(* Logix 5000 project; controller cal1615 1756-L62 rev 20.19; software revision 20.05; part 6 of 81 *)

        [13]   // Advanced Cooling Real to HMI Analog Input Recirc Fan Amps
        [14]   // Advanced Cooling Real to HMI Analog Analog Input Recirc Fan RPM
        [15]   // Advanced Cooling Real to HMI Analog Analog Input Recirc Fan Pct
        [16]   // Advanced Cooling Real to HMI Analog Input Spare
        [17]   // Advanced Cooling Real to HMI Analog Input Spare
        [24]   // Advanced Cooling Real to HMI Analog Output Hot Air Damper
        [28]   // Advanced Cooling Real to HMI Analog Output Exhaust Fan VFD Selected Speed
        [30]   // Advanced Cooling Real to HMI Analog Output Supply Fan VFD Selected Speed
        [40]   // Advanced Cooling Real to HMI Parameter TC01 Temperature Zero Offset
        [41]   // Advanced Cooling Real to HMI Parameter TC02 Temperature Zero Offset
        [42]   // Advanced Cooling Real to HMI Parameter
        [43]   // Advanced Cooling Real to HMI Parameter
        [44]   // Advanced Cooling Real to HMI Parameter PID1 NKp
        [45]   // Advanced Cooling Real to HMI Parameter PID1 Ki
        [46]   // Advanced Cooling Real to HMI Parameter PID1 Kd
        [47]   // Advanced Cooling Real to HMI Parameter PID1 Bias
        [48]   // Advanced Cooling Real to HMI Parameter PID2 Kp
        [49]   // Advanced Cooling Real to HMI Parameter PID2 Ki
        [50]   // Advanced Cooling Real to HMI Parameter PID2 Kd
        [51]   // Advanced Cooling Real to HMI Parameter PID2 Bias
        [52]   // Advanced Cooling Real to HMI Parameter Process Control High Limit
        [53]   // Advanced Cooling Real to HMI Parameter Spare
        [54]   // Advanced Cooling Real to HMI parameter Process Control Deviation
        [55]   // Advanced Cooling Real to HMI Parameter LFL Warning Level
        [56]   // Advanced Cooling Real to HMI Parameter LFL Alarm Level
        [57]   // Advanced Cooling Real to HMI Parameter Zone Shutdown Temperature
        [58]   // Advanced Cooling Real to HMI Parameter High Pressure LImit
        [59]   // Advanced Cooling Real to HMI Temperature Control Fast to Soak Control Deviation
        [60]   // Advanced Cooling Real to HMI Temperature Control Soak to Fast Control Deviation
        [61]   // Advanced Cooling Real to HMI Parameter
        [62]   // Advanced Cooling Real to HMI Parameter
        [63]   // Advanced Cooling Real to HMI Parameter
        [64]   // Advanced Cooling Real to HMI Exhaust VFD RPM Setpoint
        [65]   // Advanced Cooling Real to HMI Recirc VFD RPM Setpoint
        [67]   // Advanced Cooling Real to HMI Temperature Control Setpoint
        [68]   // Advanced Cooling Real to HMI Temperature Control manual Control Valve Setpoint
        [69]   // Advanced Cooling Real to HMI
        [70]   // Advanced Cooling Real to HMI
        [71]   // Advanced Cooling Real to HMI
        [72]   // Advanced Cooling Real to HMI Process Control Temperature
        [73]   // Advanced Cooling Real to HMI
        [74]   // Advanced Cooling Real to HMI
        [75]   // Advanced Cooling Real to HMI
        [76]   // Advanced Cooling Real to HMI
        [77]   // Advanced Cooling Real to HMI
        [78]   // Advanced Cooling Real to HMI
        [79]   // Advanced Cooling Real to HMI
   p19r01 : routine := (comment := 7);   // Advanced Cooling Main
   p19r02 : routine := (comment := -1073741761);   // Advanced Cooling Misc Control
        .WARNING.0   // Advanced Cooling Misc Control Warning 0
   p19r02_fault_exists : BOOL;
   p19r02_timer_fault : TIMER[4];   // Advanced Cooling Misc Control Fault Delay
   p19r02_timer_warning : TIMER[4] := ([0].PRE := 1500);   // Advanced Cooling Warning Delay
   p19r02_unack_fault : BOOL;   // Advanced Cooling Misc Control Unacknowledged Fault
   p19r02_unack_warning : BOOL;   // Advanced Cooling Misc Control Unacknowledged Warning
   p19r02_warning_exists : BOOL;
   p19r03 : routine := (comment := -1073741761);   // Advanced Cooling Input
   p19r03_flow_scp : SYS_SCP := (Input_Max := 100.0, Output_Max := 30840.0);   // Advanced Cooling Output Roll Cooling Flow Control
   p19r03_prs_input_max : REAL := 30840.0;
   p19r03_prs_input_min : REAL;
   p19r03_prs_output_max : REAL := 50.0;
   p19r03_prs_output_min : REAL;
   p19r03_prs_scp : SYS_SCP := (Input := 60.0, Input_Max := 100.0, Output_Max := 30840.0, Output := 18504.0);   // Advanced Cooling Output Cooling Pressure Control Valve Output
   p19r03_timer_fault : TIMER[4];   // Advanced Cooling Input
   p19r03_timer_warning : TIMER[4];   // Advanced Cooling Input
   p19r04 : routine := (comment := -1073741761);   // Advanced Cooling Output
   p19r04_timer_fault : TIMER[4];   // Advanced Cooling Output Fault Delay
   p19r04_timer_warning : TIMER[4];   // Advanced Cooling Output Warning Delay
   p19r05 : routine := (comment := -1073741761);   // Advanced Cooling Dint to HMI
   p19r05_timer_fault : TIMER[4];   // Advanced Cooing Dint to HMI
   p19r05_timer_warning : TIMER[4];   // Advanced Cooling Dint to HMI Warning Delay
   p19r06 : routine := (comment := -1073741572);   // Advanced Cooling Real to HMI
   p19r06_timer_fault : TIMER[4];   // Advanced Cooling Real to HMI Fault Delay
   p19r06_timer_warning : TIMER[4];   // Advanced Cooling Real to HMI Warning Delay
   p19r07 : routine := (comment := -1073741761);   // Advanced Cooling Alarms
   p19r07_timer_fault : TIMER[4];   // Advanced Cooling Alarms Fault Delay
   p19r07_timer_warning : TIMER[4];   // Advanced Cooling Alarms Warning Delay
   p19r08 : routine := (comment := -1073741761);   // Advanced Cooling Warnings
   p19r08_timer_fault : TIMER[4];   // Advanced Cooling Warnings Fault Delay
   p19r08_timer_warning : TIMER[4];   // Advanced Cooling Warnings Warning Delay
   p19r09 : routine := (comment := -1073741761);   // Advanced Cooling Modes
   p19r09_timer_fault : TIMER[4];   // Advanced Cooling Modes Fault Delay
   p19r09_timer_warning : TIMER[4];   // Advanced Cooling Modes Warning Delay
   p19r10 : routine := (comment := -1073741761);   // Advanced Cooling Parameters
   p19r10_timer_fault : TIMER[4];   // Advanced Cooling Parameters Fault Delay
   p19r10_timer_warning : TIMER[4];   // Advanced Cooling Parameters Warning Delay
   p19r16_pid_temp_cv : DINT;   // Advanced Cooling Temperature Control PID Control Valve
   p19r30 : routine := (comment := -1073741697);   // Advanced Cooling Temperature Control
        .FAULT.2   // Advanced Cooling Temperature Control Thermocouple Failure
        .WARNING.0   // Advanced Cooling Temperature Control Temperature Deviation Warning
        .WARNING.1   // Advanced Cooling Temperature Control Control Thermocouple 1 Failure
        .WARNING.2   // Advanced Cooling Temperature Control Control Thermocouple 2 Failure
        .WARNING.3   // Advanced Cooling Temperature Control In Manual
   p19r30_cv_man_sp : REAL := 100.0;   // Advanced Cooling Manual Control Valve Setpoint
   p19r30_pb_auto : BOOL;   // Advanced Cooling Temmperature Control PB: Zone in Auto
   p19r30_pb_manual : BOOL;   // Advanced Cooling Temmperature Control PB: Zone in Manual
   p19r30_pb_zone_off : BOOL;   // Advanced Cooling Temmperature Control PB: Zone Off
   p19r30_pb_zone_on : BOOL;   // Advanced Cooling Temmperature Control PB: Zone On
   p19r30_permissive_run : BOOL := 1;   // Advanced Cooling Temperature Control Permissive Run
   p19r30_pid_temp : PID := (CTL := -2110741376, EN := 1, CA := 1, NOBC := 1, NOZC := 1, INI := 1, OLL := 1, DVNA := 1, PVHA := 1, SP := 100.0, KP := 50.0, KI := 1.0, MAXS := 1000.0, MAXO := 100.0, UPD := 0.01, PV := 74.6, ERR := -25.400002, MAXI := 10000.0, MAXCV := 100.0, MAXTIE := 4095.0, DATA[0] := 18.470577, DATA[1] := 119.36, DATA[2] := 74.6, DATA[3] := -25.400002, DATA[4] := 100.0, DATA[5] := 0.1, DATA[6] := 0.1, DATA[7] := 0.16, DATA[8] := 50.0, DATA[9] := 1.0, DATA[11] := 50.0, DATA[12] := 1.0, DATA[15] := 1.0, DATA[16] := 0.024420025);   // Advanced Cooling Temperature Control PID
   p19r30_pid_temp_pv : DINT := 748;   // Advanced Cooling Temperature Control PID Process Variable
   p19r30_pid_temp_sp : DINT := 60;   // Advanced Cooling Temeperature Control PID Setpoint
   p19r30_request_cool : BOOL;   // Advanced Cooling Temperature Control Request Cool
   p19r30_request_manual : BOOL;   // Advanced Cooling Temperature Control Request Manual Control
   p19r30_timer_fault : TIMER[4] := ([2].PRE := 1000);   // Advanced Cooling Temperature Control Thermocouple Failure
   p19r30_timer_warning : TIMER[4] := ([0].PRE := 10000, [1].PRE := 1000, [2].PRE := 1000, [2].ACC := 1007, [2].EN := 1, [2].DN := 1, [3].PRE := 90000);   // Advanced Cooling Temperature Control Warning Delay
   p19r31 : routine := (comment := -1073741761);   // Advanced Cooling Pump
        .FAULT.0   // Advanced Cooling Pump Low Pressure
        .WARNING.0   // Advanced Cooling Pump Off
   p19r31_pb_start : BOOL;   // Advanced Cooling Pump PB: Start pump
   p19r31_pb_stop : BOOL;   // Advanced Cooling Pump PB: Stop Pump
   p19r31_request_a00 : BOOL;   // Advanced Cooling Pump Request Pressure Failure Fault
   p19r31_request_auto_run : BOOL;   // Advanced Cooling Pump Request Auto Run
   p19r31_request_manual_run : BOOL;
   p19r31_run_permissive : BOOL := 1;   // Advanced Cooling Pump Run Permissive
   p19r31_timer_fault : TIMER[4] := ([0].PRE := 5000, [1].PRE := 2000, [2].ACC := 3);   // Advanced Cooling Pump Fault Delay
   p19r31_timer_warning : TIMER[4];   // Advanced Cooling Pump Warning Delay
   p19r32 : routine := (comment := -1073741697, warning := 1, warning_ack := 1);
   p19r32_cv_man_sp : REAL;
   p19r32_pb_auto : BOOL := 1;   // Advanced Cooling Temmperature Control PB: Zone in Auto
   p19r32_pb_manual : BOOL;   // Advanced Cooling Temmperature Control PB: Zone in Manual
   p19r32_pb_zone_off : BOOL;   // Advanced Cooling Temmperature Control PB: Zone Off
   p19r32_pb_zone_on : BOOL := 1;   // Advanced Cooling Temmperature Control PB: Zone On
   p19r32_permissive_run : BOOL := 1;   // Advanced Cooling Temperature Control Permissive Run
   p19r32_pid_prs : PID := (CTL := -2110750080, EN := 1, CA := 1, NOBC := 1, NOZC := 1, INI := 1, DVPA := 1, PVHA := 1, SP := 15.0, KP := 100.0, KI := 2.0, BIAS := 3.0, MAXS := 1000.0, SO := 2.127292, MAXO := 100.0, UPD := 0.01, PV := 15.1, ERR := 0.10000038, OUT := 2.127292, MAXI := 10000.0, MAXCV := 100.0, MAXTIE := 100.0, DATA[0] := -1.8727119, DATA[1] := 24.160002, DATA[2] := 15.1, DATA[3] := 0.10000038, DATA[4] := 15.0, DATA[5] := 0.1, DATA[6] := 0.1, DATA[7] := 0.16, DATA[8] := 100.0, DATA[9] := 2.0, DATA[11] := 100.0, DATA[12] := 2.0, DATA[15] := 1.0, DATA[16] := 1.0);   // Advanced Cooling Temperature Control Pressure Control PID
        .SP   // Advanced Cooling Temperature Control Request Manual Control
        .MINCV   // Advanced Cooling Temperature Control Request Manual Control
   p19r32_pid_prs_sp : REAL := 15.0;   // Advanced Cooling Temmperature Control Pressure Setpoint
   p19r32_pid_temp_cv : REAL := 0.13189888;
   p19r32_pid_temp_pv : DINT := 149;   // Advanced Cooling Temperature Control PID Process Variable
   p19r32_request_cool : BOOL := 1;   // Advanced Cooling Temperature Control Request Cool
   p19r32_request_manual : BOOL;   // Advanced Cooling Temperature Control Request Manual Control
   p19r32_timer_fault : TIMER[4] := ([2].PRE := 1000);   // Advanced Cooling Pressure Control Fault Dwell Timer
   p19r32_timer_warning : TIMER[4] := ([1].PRE := 1000, [3].PRE := 90000);   // Advanced Cooling Pressure Control Warning Dwell Timer
   p20_acc_ctr_prs_input_max : REAL := 100.0;
   p20_acc_ctr_prs_input_min : REAL;
   p20_acc_ctr_prs_output_max : REAL := 30840.0;
   p20_acc_ctr_prs_output_min : REAL;
   p20_acc_fill_prs : REAL := 80.0;   // Upper Poly Letoff Modes A Toggle
   p20_acc_fill_prs_input_max : REAL := 100.0;
   p20_acc_fill_prs_input_min : REAL;
   p20_acc_fill_prs_output_max : REAL := 30840.0;
   p20_acc_fill_prs_output_min : REAL;
   p20_acc_fill_time_sec : REAL;   // Letoff Accumulator Fill Time
   p20_acc_input_max : REAL := 7272.0;
   p20_acc_input_min : REAL := 22340.0;
   p20_acc_output_max : REAL := 40.0;
   p20_acc_output_min : REAL;
   p20_acc_ten_prs_input_max : REAL := 100.0;
   p20_acc_ten_prs_input_min : REAL;
   p20_acc_ten_prs_output_max : REAL := 30840.0;
   p20_acc_ten_prs_output_min : REAL;
   p20_acc_tens_prs : REAL := 53.9;   // Letoff Accumulator Pressure Tension Setpoint
   p20_ai_acc_pstn : REAL;   // Letoff Analog Input Accumulator Position
   p20_ai_lc01 : REAL := 2.7937975;   // Letoff Analog Input Line Tension Load Cell Splicer
   p20_ai_letoff_dia : REAL := 53.379654;   // Letoff Analog Inputs Letoff Roll Diameter [in]
   p20_ai_lo_turret_amps : REAL;   // Letoff Inputs Letoff Turret VFD Amps
   p20_ai_lo_turret_hz : REAL := -3.8146973e-06;   // Letoff Inputs Letoff Turret VFD Hz
   p20_ai_lo_turret_speed : REAL;
   p20_ai_loa_speed : REAL;   // Letoff Inputs Letoff A VFD Surface Speed
   p20_ai_lob_speed : REAL;   // Letoff Inputs Letoff A Speed
   p20_ao_acc_ctr_prs : REAL := 10.0;   // Letoff Analog Output Accumulator Counter Pressure
   p20_ao_acc_fill_prs : REAL := 32.0;   // Letoff Analog Output Accumulator Fill Pressure
   p20_ao_acc_ten_prs : REAL := 32.0;   // Letoff Analog Output Accumulator Tension Pressure
   p20_ao_lo_turret_selected_speed : REAL;   // Letoff Letoff Turret VFD Selected Speed
   p20_ao_loa_selected_speed : REAL;   // Letoff Output Selected Speed
   p20_ao_loa_torque : REAL := 80.0;
   p20_ao_lob_selected_speed : REAL;   // Letoff Letoff B VFD Selected Speed
   p20_ao_lob_torque : REAL := 80.0;
   p20_di_acc_door_open : BOOL;
   p20_di_acc_empty : BOOL := 1;   // Letoff Digital Input Letoff Accumulator Empty Position
   p20_di_acc_full : BOOL;   // Letoff Digital Input Letoff Accumulator Full Control Position
   p20_di_clutch_prs_ok : BOOL;   // Letoff Modes Accumulator Position Mode
   p20_di_lfr_jog_fwd : BOOL;   // Letoff Digital Input PB: Feedroll Jog Forward
   p20_di_lfr_jog_rev : BOOL;   // Letoff Digital Input PB: Feedroll Jog Reverse
   p20_di_lfr_nip_close : BOOL;   // Letoff Digital Input PB: Feedroll Nip Roll Close
   p20_di_lo_turret : acs800_di_normal := (ready := 1, ctrl_from_net := 1, ref_from_net := 1);   // Letoff Letoff Turret VFD Drive Inputs
   p20_di_lo_turret_therm : BOOL := 1;   // Letoff Input Letoff Turret Motor Temp Ok
   p20_di_loa_active : BOOL := 1;   // Letoff Digital Input Letoff A Active
   p20_di_loa_brake : BOOL := 1;   // Letoff Input Letoff A Brake Temperature Ok
   p20_di_loa_fwd_dir : BOOL := 1;   // Letoff Digital Inputs PB: Letoff A Jog FWD
   p20_di_loa_jog : BOOL;   // Letoff Digital Inputs PB: Letoff A Jog REV
   p20_di_loa_start : BOOL;   // Letoff Digital Input PB: Letoff A Start
   p20_di_loa_stop : BOOL := 1;   // Letoff Digital Input PB: Letoff A Stop Stop = 0
   p20_di_loa_temp : BOOL := 1;   // Letoff Input Letoff A Motor Temperature Ok
   p20_di_lob_brake_thermostat : BOOL := 1;   // Letoff Input Letoff B Brake Temperature OK
   p20_di_lob_fwd_dir : BOOL := 1;   // Letoff Digital Inputs PB: Letoff B Jog FWD
   p20_di_lob_jog : BOOL;   // Letoff Digital Inputs PB: Letoff B Jog REV
   p20_di_lob_motor_thermostat : BOOL := 1;   // Letoff Input Letoff B Motor Temperature Ok
   p20_di_lob_start : BOOL;   // Letoff Digital Input PB: Letoff B Start
   p20_di_lob_stop : BOOL := 1;   // Letoff Digital Input PB: Letoff B Stop
   p20_di_lof_acc_fill : BOOL;   // Letoff Digital Input PB: Accumulator Fill
   p20_di_turret_fwd : BOOL;   // Letoff Digital Inputs PB: Turret FWD
   p20_di_turret_pos : BOOL := 1;   // Letoff Digital Inputs PX: Turret in Position
   p20_di_turret_rev : BOOL;   // Letoff Digital Inputs PB: Turret REV
   p20_dia_input_max : REAL := 30959.0;
   p20_dia_input_min : REAL := 100.0;
   p20_dia_output_max : REAL := 53.0;
   p20_dia_output_min : REAL := 5.0;
   p20_dint_to_hmi : DINT[16] := ([0] := 37, [1] := 7401712, [4] := 33, [6] := 131072, [7] := 1);   // Letoff Dint to HMI
        [0].0   // Letoff Dint to HMI Letoff A Active
        [0].1   // Letoff Dint to HMI Letoff B Active
        [0].2   // Letoff Dint to HMI Letoff Turret in Position
        [0].4   // Letoff Dint to HMI Letoff Accumulator Full Control Position
        [0].5   // Letoff Dint to HMI Letoff Accumulator Empty Control Position
        [0].8   // Letoff Dint to HMI Accumulator Auto Mode
        [1].0   // Letoff Dint to HMI Letoff A VFD Faulted
        [1].1   // Letoff Dint to HMI Letoff A VFD Warning
        [1].2   // Letoff Dint to HMI Letoff A VFD Running Forward
        [1].3   // Letoff Dint to HMI Letoff A VFD Running Reverse
        [1].4   // Letoff Dint to HMI Letoff A VFD Ready
        [1].5   // Letoff Dint to HMI Letoff A VFD Control From Net
        [1].6   // Letoff Dint to HMI Letoff A VFD Reference From Net
        [1].7   // Letoff Dint to HMI Letoff A VFD At Reference
        [1].8   // Letoff Dint to HMI Letoff B VFD Faulted
        [1].9   // Letoff Dint to HMI Letoff B VFD Warning
        [1].10   // Letoff Dint to HMI Letoff B VFD Running Forward
        [1].11   // Letoff Dint to HMI Letoff B VFD Running Reverse
        [1].12   // Letoff Dint to HMI Letoff B VFD Ready
        [1].13   // Letoff Dint to HMI Letoff B VFD Control From Net
        [1].14   // Letoff Dint to HMI Letoff B VFD Reference From Net
        [1].15   // Letoff Dint to HMI Letoff B VFD At Reference
        [1].16   // Letoff Dint to HMI Letoff Turret VFD Faulted
        [1].17   // Letoff Dint to HMI Letoff Turret VFD Warning
        [1].18   // Letoff Dint to HMI Letoff Turret VFD Running Forward
        [1].19   // Letoff Dint to HMI Letoff Turret VFD Running Reverse
        [1].20   // Letoff Dint to HMI Letoff Turret VFD Ready
        [1].21   // Letoff Dint to HMI Letoff Turret VFD Control from Net
        [1].22   // Letoff Dint to HMI Letoff Turret VFD Reference From Net
        [1].23   // Letoff Dint to HMI Letoff Turret VFD At Reference
        [2].0   // Letoff Alarms A00: Letoff A VFD Faulted
        [2].1   // Letoff Alarms A01:
        [2].2   // Letoff Alarms A02: Letoff A VFD Drive Not Ready
        [2].3   // Letoff Alarms A03: Letoff A VFD Drive Not in Remote Mode
        [2].4   // Letoff Alarms A04 :Letoff A VFD Motor Temperature
        [2].5   // Letoff Alarms A05: Letoff A VFD Brake Temperature
        [2].6   // Letoff Alarms A06: Letoff B VFD Drive Faulted
        [2].7   // Letoff Alarms A07:
        [2].8   // Letoff Alarms A08: Letoff B VFD Drive Not Ready
        [2].9   // Letoff Alarms A09: Letoff B VFD Drive Not in Remote Mode
        [2].10   // Letoff Alarms A10: Letoff B VFD Motor Temperature
        [2].11   // Letoff Alarms A11: Letoff B VFD Brake Temperature
        [2].12   // Letoff Alarms A12: Letoff Turret VFD Drive Faulted
        [2].13   // Letoff Alarms A13:
        [2].14   // Letoff Alarms A14: Letoff Turret VFD Drive not Ready
        [2].15   // Letoff Alarms A15: Letoff Turret VFD Drive not in Remote Mode
        [2].16   // Letoff Alarms A16:
        [2].17   // Letoff Alarms A17: Letoff Turret VFD Motor Temperature
        [2].18   // Letoff Alarms A18:
        [2].19   // Letoff Alarms A19:
        [2].20   // Letoff Alarms A20:
        [2].21   // Letoff Alarms A21:
        [2].22   // Letoff Alarms A22:
        [2].23   // Letoff Alarms A23:
        [2].24   // Letoff Alarms A24:
        [2].25   // Letoff Alarms A25:
        [2].26   // Letoff Alarms A26:
        [2].27   // Letoff Alarms A27:
        [2].28   // Letoff Alarms A28:
        [2].29   // Letoff Alarms A29:
        [2].30   // Letoff Alarms A30:
        [2].31   // Letoff Alarms A31:
        [4].0   // Letoff Warnings W00: Letoff A VFD Drive Warning
        [4].1   // Letoff Warnings W01: Letoff B Drive Warning
        [4].2   // Letoff Warnings W02: Letoff Turret VFD Drive Warning
        [4].3   // Letoff Warnings W03: Index Not Complete
        [4].4   // Letoff Warnings W04: No Letoff Selected
        [4].5   // Letoff Warnings W05:
        [4].6   // Letoff Warnings W06:
        [4].7   // Letoff Warnings W07:
        [4].8   // Letoff Warnings W08:
        [4].9   // Letoff Warnings W09:
        [4].10   // Letoff Warnings W10:
        [4].11   // Letoff Warnings W11:
        [4].12   // Letoff Warnings W12:
        [4].13   // Letoff Warnings W13:
        [4].14   // Letoff Warnings W14:
        [4].15   // Letoff Warnings W15:
        [4].16   // Letoff Warnings W16:
        [4].17   // Letoff Warnings W17:
        [4].18   // Letoff Warnings W18:
        [4].19   // Letoff Warnings W19:
        [4].20   // Letoff Warnings W20:
        [4].21   // Letoff Warnings W21:
        [4].22   // Letoff Warnings W22:
        [4].23   // Letoff Warnings W23:
        [4].24   // Letoff Warnings W24:
        [4].25   // Letoff Warnings W25:
        [4].26   // Letoff Warnings W26:
        [4].27   // Letoff Warnings W27:
        [4].28   // Letoff Warnings W28:
        [4].29   // Letoff Warnings W29:
        [4].30   // Letoff Warnings W30:
        [4].31   // Letoff Warnings W31:
   p20_do_acc_enable_tension : BOOL := 1;   // Letoff Digital Output Enable Accumulator Lift Tension
   p20_do_acc_high_prs : BOOL;   // Letoff Digital Output Enable Accumulator Lift Pressure
   p20_do_close_nip : BOOL;   // Letoff Digital Output Feedroll Roll Nip Close
   p20_do_enable_lfr_fwd : BOOL;   // Letoff Digital Output Letoff Accumulator Feedroll Forward
   p20_do_enable_lfr_rev : BOOL;   // Letoff Digital Output Letoff Accumulator Feedroll Reverse
   p20_do_engage_lfr_clutch : BOOL;   // Letoff Digital Output Engage Letoff Accumulator Feedroll Clutch
   p20_do_wdr_turret : acs800_do_normal;
        .FORWARD   // Letoff Letoff Turret VFD Request Jog FWD
        .REVERSE   // Letoff Letoff Turret VFD Request Jog REV
        .FAULT_RESET   // Letoff Letoff Turret VFD Fault Reset
   p20_lc_input_max : REAL := 10000.0;
   p20_lc_input_min : REAL;   // Letoff Analog Input
   p20_lc_output_max : REAL := 153.4;
   p20_lc_output_min : REAL;
   p20_loa_ai_amps : REAL;   // Letoff Inputs Letoff A VFD Amps
   p20_loa_ai_hz : REAL := 3.8146973e-06;   // Letoff Inputs Letoff A Hz
   p20_loa_ai_rpm : REAL;
   p20_loa_ai_torque : REAL;
   p20_loa_footage_input_max : REAL := 9000.0;
   p20_loa_footage_input_min : REAL;
   p20_loa_footage_output_max : REAL := 9000.0;
   p20_loa_footage_output_min : REAL;
   p20_lob_ai_amps : REAL;   // Letoff Inputs Letoff B VFD Amps
   p20_lob_ai_hz : REAL := -3.8146973e-06;   // Letoff Inputs Letoff B VFD Hz
   p20_lob_ai_rpm : REAL;
   p20_lob_ai_torque : REAL;
   p20_lob_footage_input_max : REAL := 9000.0;
   p20_lob_footage_input_min : REAL;
   p20_lob_footage_output_max : REAL := 9000.0;
   p20_lob_footage_output_min : REAL;
   p20_param_acc_auto_fill : REAL := 10.0;
   p20_param_acc_ctr_prs : REAL := 10.0;   // Letoff Parameter Carriage Counter Pressure Setpoint
   p20_param_acc_empty_prs : REAL := 32.0;
   p20_param_acc_fast_accel : REAL := 100.0;
   p20_param_acc_fast_decel : REAL := 100.0;
   p20_param_acc_fill_ctr_prs : REAL := 5.0;
   p20_param_acc_high_prs : REAL := 10.0;   // Letoff Parameter High Pressure Setpoint
   p20_param_acc_init_high_prs : REAL := 1.5;
   p20_param_acc_init_low_prs : REAL := 1.0;
   p20_param_acc_init_prs : REAL := 1.0;   // Letoff Accumulator Initial Pressure for Ramp
   p20_param_acc_med_accel : REAL := 1.0;
   p20_param_acc_med_decel : REAL := 1.0;
   p20_param_acc_pid_accel : REAL := 2.0;
   p20_param_acc_pid_decel : REAL := 2.0;
   p20_param_acc_pos_prs : REAL := 10.0;
   p20_param_acc_slow_accel : REAL := 0.5;
   p20_param_acc_slow_decel : REAL := 0.5;
   p20_param_empty_pct : REAL := 0.5;
   p20_param_high_accel_rate : REAL := 100.0;
   p20_param_high_ctrl_pct : REAL := 60.0;   // Letoff Parameter High Accumulator Control Position
   p20_param_high_decel_rate : REAL := 100.0;
   p20_param_high_ki : REAL := 0.01;
   p20_param_high_kp : REAL := 1000.0;
   p20_param_high_low_ctrl_pct : REAL := 10.0;   // Letoff Accumulator High Control Position Low Limit
   p20_param_high_upd : REAL := 0.01;
   p20_param_jog_accel_rate : REAL := 10.0;
   p20_param_jog_decel_rate : REAL := 10.0;
   p20_param_letoff_jog_speed : REAL := 20.0;
   p20_param_lo_turret_gear_ratio : REAL := 1200.0;
   p20_param_lo_turret_index_speed : REAL := 8.0;
   p20_param_loa_gear_ratio : REAL := 50.86;
   p20_param_lob_gear_ratio : REAL := 50.86;
   p20_param_lof_fast_fill : REAL := 50.0;
   p20_param_lof_slow_fill : REAL := 40.0;
   p20_param_lof_stop_fill : REAL := 30.0;
   p20_param_low_ctrl_pct : REAL := 7.0;   // Letoff Parameter Low Accumulator Control Position
   p20_param_low_low_ctrl_pct : REAL := 2.0;
   p20_param_norm_accel_rate : REAL := 2.0;
   p20_param_norm_decel_rate : REAL := 20.0;   // Letoff Parameter Letoff A Decel Rate
   p20_param_prs_accel_rate : REAL := 1.0;   // Letoff Accumulator Accel/Decel Ramp Accel Rate
   p20_param_prs_decel_rate : REAL := 1.0;   // Letoff Accumulator Accel/Decel Ramp Decel Rate
   p20_param_run_torque : REAL := 80.0;
   p20_real_to_hmi : REAL[112] := ([0] := 2.8150334, [1] := 53.348545, [8] := 3.8146973e-06, [14] := -3.8146973e-06, [15] := 65.0, [20] := -3.8146973e-06, [21] := 8541.531, [22] := 1.7456055, [25] := 10.0, [26] := 32.0, [27] := 32.0, [40] := 1.1, [41] := 2.0);   // Letoff Real to HMI
        [0]   // Letoff Real to HMI Letoff Tension
        [1]   // Letoff Real to HMI Letoff Diameter
        [2]   // Letoff Real to HMI Letoff Accumulator Position
        [6]   // Letoff Real to HMI Letoff A Speed
        [7]   // Letoff Real to HMI Letoff A Amps
        [8]   // Letoff Real to HMI Letoff A Hertz
        [12]   // Letoff Real to HMI Letoff B Speed
        [13]   // Letoff Real to HMI Letoff B Amps
        [14]   // Letoff Real to HMI Letoff B Hertz
        [18]   // Letoff Real to HMI Letoff Turret Speed
        [19]   // Letoff Real to HMI Letoff Turret Amps
        [20]   // Letoff Real to HMI Letoff Turret Hertz
   p20_request_run_index_dir : BOOL;   // Letoff Letoff Turret Request Run Index Direction
   p20_request_run_index_rev_dir : BOOL;   // Letoff Letoff Turret Request Run Index Reverse Direction
   p20_vfd_di_loa : acs800_di_normal := (ready := 1, ctrl_from_net := 1, ref_from_net := 1, at_reference := 1);   // Letoff A VFD Inputs
   p20_vfd_di_lob : acs800_di_normal := (ready := 1, ctrl_from_net := 1, ref_from_net := 1, at_reference := 1);   // Letoff B VFD Inputs
   p20_vfd_do_loa : acs800_do_normal;   // Letoff A VFD Outputs
   p20_vfd_do_lob : acs800_do_normal;   // Letoff B VFD Outputs
   p20_zero_tension_prs : REAL := 38.0;
   p20r01 : routine := (comment := 7);   // Letoff Main
   p20r02 : routine := (comment := -1073741761);   // Letoff Misc Control
        .UNACK_FAULT   // Letoff Misc Control Unacknowledged Faults Exists
        .UNACK_WARNING   // Letoff Misc Control Unacknowledged Warning Exists
   p20r02_fault_exists : BOOL;
   p20r02_letoff_dia_ft : REAL := 2.1791723;   // Letoff Misc Control Letoff Diameter [ft]
   p20r02_letoff_selection_dwell : TIMER := (PRE := 60000, EN := 1, DN := 1);
   p20r02_timer_fault : TIMER[4];   // Letoff Misc Control Fault Delay
   p20r02_timer_warning : TIMER[4];   // Letoff Misc Control Warning Delay
   p20r02_unack_fault : BOOL;   // Letoff Misc Control Unacknowledge Fault Exists
   p20r02_unack_warning : BOOL := 1;   // Letoff Misc Control Unacknowledge Warning Exists
   p20r02_warning_exists : BOOL := 1;
   p20r03 : routine := (comment := -1073741761);   // Letoff Input
        .UNACK_FAULT   // Letoff Input Unacknowledged Faults Exists
        .UNACK_WARNING   // Letoff Input Unacknowledged Warning Exists
   p20r03_accumulator_pct_scp : SYS_SCP := (Input := 22376.0, Input_Min := 22340.0, Input_Max := 7272.0, Output_Max := 100.0);   // Letoff Analog Inputs Accumulator Position 0-100%
   p20r03_accumulator_scp : SYS_SCP := (Input := 22360.0, Input_Min := 22340.0, Input_Max := 7272.0, Output_Max := 40.0);   // Letoff Analog Inputs Accumulator Position 0-63 in
   p20r03_distance_to_core : REAL := 32.55;
   p20r03_lo_radius : REAL := 26.689827;   // Letoff Analog Inputs Letoff Roll Radius
   p20r03_lo_turret_speed_fb : SYS_RPM_TO_SPEED := (IN_gear_ratio := 1200.0, IN_roll_diameter := 3.2);   // Letoff Inputs Letoff Turret Speed Feedback
   p20r03_loa_distance_to_core : REAL := 32.55;
   p20r03_Loa_footage_scp : SYS_SCP := (Input := 8541.955, Input_Max := 9000.0, Output_Max := 9000.0, Output := 8541.955);   // Letoff Analog Inputs Letoff A Footage Counter Scaling
   p20r03_loa_speed_fb : SYS_RPM_TO_SPEED := (IN_gear_ratio := 50.86, IN_roll_diameter := 2.1791723);   // Letoff Inputs Letoff A VFD Speed Feedback SCP
   p20r03_load_cell : SYS_SCP := (Input := 185.85449, Input_Max := 10000.0, Output_Max := 153.4, Output := 2.8510077);   // Letoff Analog Input Load Cell Scaling 0-(2*150lbs)
   p20r03_lob_distance_to_core : REAL := 32.8;
   p20r03_Lob_footage_scp : SYS_SCP := (Input := 1.7456055, Input_Max := 9000.0, Output_Max := 9000.0, Output := 1.7456055);   // Letoff Analog Inputs Letoff B Footage Counter Scaling
   p20r03_lob_speed_fb : SYS_RPM_TO_SPEED := (IN_gear_ratio := 50.86, IN_roll_diameter := 2.1791723);   // Letoff Inputs Letoff B VFD Speed Feedback SCP
   p20r03_sensor_input : REAL := 5.8757267;
   p20r03_sensor_scp : SYS_SCP := (Input := 663.0, Input_Min := 100.0, Input_Max := 30959.0, Output_Min := 5.0, Output_Max := 53.0, Output := 5.8757267);   // Letoff Analog Input Sensor Scaling
   p20r03_timer_fault : TIMER[4];   // Letoff Input Fault Delay
   p20r03_timer_warning : TIMER[4];   // Letoff Input Warning Delay
   p20r04 : routine := (comment := -1073741761);   // Letoff Ouput
        .UNACK_FAULT   // Letoff Output Unacknowledged Faults Exists
        .UNACK_WARNING   // Letoff Output Unacknowledged Warning Exists
   p20r04_acc_ctr_prs : SYS_SCP := (Input := 10.0, Input_Max := 100.0, Output_Max := 30840.0, Output := 3084.0);   // Letoff Analog Outputs Accumulator Counter Pressure
   p20r04_acc_fill_prs : SYS_SCP := (Input := 32.0, Input_Max := 100.0, Output_Max := 30840.0, Output := 9868.8);   // Letoff Analog Output Accumulator Fill Pressure
   p20r04_acc_ten_prs : SYS_SCP := (Input := 32.0, Input_Max := 100.0, Output_Max := 30840.0, Output := 9868.8);   // Letoff Analog Output Accumulator Tension Pressure
   p20r04_lo_turret_speed_to_vfd : SYS_SPEED_TO_VFD := (IN_gear_ratio := 1200.0, IN_roll_diameter := 3.2);   // Letoff Outputs Letoff Turret Speed
   p20r04_loa_speed_to_vfd : SYS_SPEED_TO_VFD := (IN_gear_ratio := 50.86, IN_roll_diameter := 2.1791723);   // Letoff Outputs Letoff A Speed
   p20r04_lob_speed_to_vfd : SYS_SPEED_TO_VFD := (IN_gear_ratio := 50.86, IN_roll_diameter := 2.1791723);   // Letoff Outputs Letoff B Speed
   p20r04_timer_fault : TIMER[4];   // Letoff Output Fault Delay
   p20r04_timer_warning : TIMER[4];   // Letoff Output Warning Delay
   p20r05 : routine := (comment := -1073741761);   // Letoff Dint to HMI
        .UNACK_FAULT   // Letoff Dint to HMI Unacknowledged Faults Exists
        .UNACK_WARNING   // Letoff Dint to HMI Unacknowledged Warning Exists
   p20r05_timer_fault : TIMER[4];   // Letoff Dint to HMI Fault Delay
   p20r05_timer_warning : TIMER[4];   // Letoff Dint to HMI Warning Delay
   p20r06 : routine := (comment := -1073741572);   // Letoff Real to HMI
        .UNACK_FAULT   // Letoff Real to HMI Unacknowledged Faults Exists
        .UNACK_WARNING   // Letoff Real to HMI Unacknowledged Warning Exists
   p20r06_ave_lc : REAL := 2.8223236;
   p20r06_lc_ave_ctrl : CONTROL := (LEN := 19);
   p20r06_lc_buffer : REAL[20] := ([0] := 2.8269193, [1] := 2.7877753, [2] := 2.8510077, [3] := 2.8449857, [4] := 2.7937975, [5] := 2.8419745, [6] := 2.742609, [7] := 2.8510077, [8] := 2.7968085, [9] := 2.823908, [10] := 2.814875, [11] := 2.781753, [12] := 2.8600411, [13] := 2.8088527, [14] := 2.8359525, [15] := 2.820897, [16] := 2.8359525, [17] := 2.7998195, [18] := 2.7877753, [19] := 2.8449857);
   p20r06_lc_ctrl : CONTROL := (LEN := 20, POS := 20, DN := 1);
   p20r06_sample_timer : TIMER := (PRE := 200, ACC := 132, EN := 1, TT := 1);
   p20r06_timer_fault : TIMER[4];   // Letoff Real to HMI Fault Delay
   p20r06_timer_warning : TIMER[4];   // Letoff Real to HMI Warning Delay
   p20r06_unload : DINT := 3;
   p20r07 : routine := (comment := -1073741761);   // Letoff Alarms
        .UNACK_FAULT   // Letoff Alarms Unacknowledged Faults Exists
        .UNACK_WARNING   // Letoff Alarms Unacknowledged Warning Exists
   p20r07_timer_fault : TIMER[4];   // Letoff Alarms Fault Delay
   p20r07_timer_warning : TIMER[4];   // Letoff Alarms Warning Delay
   p20r08 : routine := (comment := -1073741761);   // Letoff Warnings
        .UNACK_FAULT   // Letoff Warnings Unacknowledged Faults Exists
        .UNACK_WARNING   // Letoff Warnings Unacknowledged Warning Exists
   p20r08_timer_fault : TIMER[4];   // Letoff Warnings Fault Delay
   p20r08_timer_warning : TIMER[4];   // Letoff Warnings Warning Delay
   p20r09 : routine := (comment := -1073741761, fault := 1, fault_ack := 1);   // Letoff Modes
        .UNACK_FAULT   // Letoff Modes Unacknowledged Faults Exists
        .UNACK_WARNING   // Letoff Modes Unacknowledged Warning Exists
   p20r09_acc_toggle : SYS_Toggle;   // Letoff Modes Accumulator Auto
   p20r09_accumulator_auto : BOOL;   // Letoff Modes Accumulator Auto Mode
   p20r09_letoff_a_active : BOOL := 1;   // Letoff Modes Letoff A Active
   p20r09_timer_fault : TIMER[4];   // Letoff Modes Fault Delay
   p20r09_timer_warning : TIMER[4];   // Letoff Modes Warning Delay
   p20r10 : routine := (comment := -1073739969, oneshot := 1);   // Letoff Letoff Tension Control
        .WARNING.1   // Letoff Letoff Brake High Tension
        .UNACK_FAULT   // Letoff Tension Control Unacknowledged Faults Exists
        .UNACK_WARNING   // Letoff Tension Control Unacknowledged Warning Exists
   p20r10_param_acc_full_psn : REAL := 100.0;
   p20r10_param_fill_gain : REAL := 0.0198;
   p20r10_param_normal_gain : REAL := 0.01;
   p20r10_param_psn_gain : REAL := 0.01;   // Letoff Letoff Tension Control Tension Gain
   p20r10_pid_psn : PID := (CTL := -2078243968, EN := 1, SWM := 1, NOBC := 1, INI := 1, DVPA := 1, PVLA := 1, PVHA := 1, SP := 100.0, KP := 250.0, BIAS := 5.0, MAXS := 100.0, SO := 100.0, MAXO := 100.0, UPD := 0.01, ERR := 100.0, OUT := 100.0, MAXI := 100.0, MAXCV := 100.0, MAXTIE := 100.0, DATA[3] := 100.0, DATA[4] := 100.0, DATA[5] := 1.0, DATA[6] := 1.0, DATA[7] := 0.16, DATA[8] := 250.0, DATA[11] := 250.0, DATA[15] := 1.0, DATA[16] := 1.0);   // Letoff Letoff Position Control PID
   p20r10_pid_psn_cv : REAL := 100.0;
   p20r10_pid_psn_pv : REAL;   // Letoff Letoff Positon Control PID Process Value
   p20r10_pid_tens : PID := (CTL := -2078244224, EN := 1, SWM := 1, NOBC := 1, INI := 1, DVPA := 1, PVHA := 1, SP := 15.0, KP := 1.1, KI := 2.0, MAXS := 500.0, SO := 65.0, MAXO := 100.0, UPD := 0.01, PV := 2.8329413, ERR := 12.167059, OUT := 65.0, MAXI := 500.0, MAXCV := 100.0, MAXTIE := 100.0, DATA[0] := 62.323246, DATA[1] := -9.0654125, DATA[2] := 2.8329413, DATA[3] := 12.167059, DATA[4] := 15.0, DATA[5] := 0.2, DATA[6] := 1.0, DATA[7] := 0.16, DATA[8] := 1.1, DATA[9] := 2.0, DATA[11] := 1.1, DATA[12] := 2.0, DATA[15] := 1.0, DATA[16] := 1.0);   // Letoff Letoff Speed Control Tension PID
   p20r10_pid_tens_cv : REAL := 65.0;   // Letoff Letoff Speed Control Control Value CV
   p20r10_pid_tens_pv : REAL := 2.8449857;   // Letoff Letoff Tension Control PID Process Value
   p20r10_run_permissive : BOOL := 1;   // Letoff Letoff Tension Control Run Permissive
   p20r10_speed_offset : REAL := 0.5;   // Letoff Letoff Speed Control Speed Offset
   p20r10_speed_offset_psn : REAL := 0.5;   // Letoff Letoff Speed Control Position PID Speed Offset
   p20r10_speed_offset_tens : REAL := -0.14999999;   // Letoff Letoff Speed Control Tension PID Speed Offset
   p20r10_tension_request : BOOL;   // Letoff Letoff Tension Control Tension Control Request
   p20r10_timer : TIMER[2] := ([0].PRE := 10, [0].ACC := 33, [0].EN := 1, [0].DN := 1);   // Letoff Letoff Tension Control PID Condition
   p20r10_timer_fault : TIMER[4];   // Letoff Fault Delay
   p20r10_timer_warning : TIMER[4];   // Letoff Warning Delay
   p20r11 : routine := (comment := -1073741793);   // Letoff Feedroll
        .UNACK_FAULT   // Letoff Feedroll Unacknowledged Faults Exists
        .UNACK_WARNING   // Letoff Feedroll Unacknowledged Warning Exists
   p20r11_manual_open_nip : BOOL;   // Letoff Feedroll Request Manual Open Nip
   p20r11_nip_close_dwell : TIMER := (PRE := 1000);
   p20r11_permissive_jog : BOOL;   // Letoff Feedroll Permissive Jog
   p20r11_permissive_run : BOOL;   // Letoff Feedroll Permissive Run
   p20r11_request_close_nip : BOOL;   // Letoff Feedroll Request Close Feedroll Nip Roll
   p20r11_request_jog_fwd : BOOL;   // Letoff Feedroll Request Jog Forward
   p20r11_request_jog_rev : BOOL;   // Letoff Feedroll Request Jog Reverse
   p20r11_timer_clutch_off : TIMER := (PRE := 300, ACC := 300);   // Letoff Feedroll Clutch Off Delay
   p20r11_timer_clutch_on : TIMER := (PRE := 300);   // Letoff Feedroll Clutch On Delay
   p20r11_timer_fault : TIMER[4];   // Letoff Feedroll Fault Delay
   p20r11_timer_warning : TIMER[4];   // Letoff Feedroll Warning Delay
   p20r13 : routine := (comment := -1073741761, oneshot := 1);   // Letoff Accum Control
        .FAULT.1   // Letoff Accumulator Empty Position Calibration Error
        .WARNING.0   // Letoff Accum Control Accumulator Empty
        .WARNING.1   // Letoff Accum Control Accumulator Full
        .WARNING.2   // Letoff Accumulator High Position Calibration Error
        .WARNING.3   // Letoff Accumulator Empty Position Calibration Error
        .UNACK_FAULT   // Letoff Accumulator Unacknowledged Faults Exists
        .UNACK_WARNING   // Letoff Accumulator Unacknowledged Warning Exists
   p20r13_acc_top_pos : REAL := 99.7;   // Upper Poly Letoff Modes Letoff B Tension Mode
   p20r13_ai_acc_pct : REAL;   // Letoff Accumulator Pct Full
   p20r13_ai_loa_footage_ft : REAL := 8541.248;
   p20r13_ai_lob_footage_ft : REAL := 1.7456055;
   p20r13_enc : SYS_ENC := (IN_State := 3, OUT_Status := 1);   // Letoff Accumulator Encoder
   p20r13_ramp_tension_pressure : SYS_ACC_DEC_RAMP := (IN_selected_line_speed := 32.0, IN_param_master_accel_rate := 1.0, IN_param_master_decel_rate := 1.0, IN_last_scan_s := 0.032382);   // Letoff Accumulator Tension Pressure Ramp
        .DATA.0   // Digital Input Zone 3 Recirculation Fan Rotating
        .DATA.1   // Digital Input Zone 3 Exhaust Fan Rotating
        .DATA.2   // Digital Input Zone 3 Spare
        .DATA.3   // Digital Input Zone 3 Spare
        .DATA.4   // Digital Input Zone 3 Spare
        .DATA.5   // Digital Input Zone 3 Spare
        .DATA.6   // Digital Input Zone 3 Spare
        .DATA.7   // Digital Input Zone 3 Spare
        .DATA.8   // Digital Input Rope Switch 1 Active
        .DATA.9   // Digital Input Rope Switch 2 Active
        .DATA.10   // Digital Input Rope Switch 3 Active
        .DATA.11   // Digital Input Rope Switch 4 Active
        .DATA.12   // Digital Input Rope Switch 5 Active
        .DATA.13   // Digital Input Rope Switch 6 Active
        .DATA.14   // Digital Input Rope Switch 7 Active
        .DATA.15   // Digital Input Rope Switch 8 Active
   p20r13_request_fill : BOOL;   // Letoff Accumulator Request Fill
   p20r13_selected_pressure : REAL := 32.0;   // Letoff Accumulator Selected Pressure
   p20r13_state : DINT := 3;   // Letoff Accumulator State
        .0   // Letoff Accumulator State One Set per Scan
        .1   // Letoff Accumulator State 1 Idle/Control to Low Position
        .2   // Letoff Accumulator State 2 Fill Request
        .3   // Letoff Accumulator State 3 Ramp Tension Pressure
        .4   // Letoff Accumulator State 4 Fill to Full Position
        .5   // Letoff Accumulator State 5 Control to Top Hard Stop
        .6   // Letoff Accumulator State 6 Payout Request
        .7   // Letoff Accumulator State 7 Payout to Empty
        .8   // Letoff Accumulator State 8 Lower Limit Reached
        .9   // Letoff Accumulator State 9 Complete
        .10   // Letoff Accumulator State 10 Position Mode Fill Request
        .11   // Letoff Accumulator State 11 Position Mode Fill to Full Position
        .12   // Letoff Accumulator State 12 Position Mode Control to Top Position
   p20r13_status : DINT := 1;   // Letoff Accumulator Fill Status
   p20r13_timer_fault : TIMER[4];   // Letoff Accum Control Fault Delay
   p20r13_timer_warning : TIMER[4];   // Letoff Accum Control Warning Delay
   p20r14 : routine := (comment := -1073741761, fault := 1, fault_ack := 1);   // Letoff Accumulator Fill Pressure
        .UNACK_FAULT   // Letoff Accumulator Fill Pressure Unacknowledged Faults Exists
        .UNACK_WARNING   // Letoff Accumulator Fill Pressure Unacknowledged Warning Exists
   p20r14_acc_request_tension_ctrl : BOOL;   // Letoff Accumulator Fill Pressure Request Tension Control
   p20r15 : routine := (comment := -536870793, warning := 1, unack_warning := 1);   // Letoff Letoff A VFD
        .FAULT.0   // Letoff Letoff A VFD Drive Faulted
        .FAULT.2   // Letoff Letoff A VFD Drive Not Ready
        .FAULT.3   // Letoff Letoff A VFD Drive Not in Remote Mode
        .FAULT.4   // Letoff Letoff A VFD Motor Temperature
        .FAULT.5   // Letoff Letoff A Brake Temperature
        .WARNING   // Letoff Letoff A VFD
        .WARNING.0   // Letoff Letoff A VFD Warning
        .UNACK_FAULT   // Letoff Letoff A VFD Unacknowledged Faults Exists
        .UNACK_WARNING   // Letoff Letoff A VFD Unacknowledged Warning Exists
   p20r15_loa_accel : REAL := 100.0;   // Letoff Letoff A VFD Accel Rate ORG: 100
   p20r15_loa_accel_decel_ramp : SYS_ACC_DEC_RAMP := (IN_param_master_accel_rate := 100.0, IN_param_master_decel_rate := 100.0, IN_last_scan_s := 0.033042);   // Letoff Letoff A VFD Accel Decel Ramp
   p20r15_loa_decel : REAL := 100.0;   // Letoff Letoff A VFD Decel Rate ORG: 20
   p20r15_loa_on : BOOL := 1;   // Letoff Letoff A VFD On
   p20r15_loa_selected_speed : REAL;   // Letoff Letoff A VFD Selected Speed
   p20r15_permissive_run : BOOL := 1;   // Letoff Letoff A VFD Permissive Run
   p20r15_request_jog_fwd : BOOL;   // Letoff Letoff A VFD Request Jog FWD
   p20r15_request_jog_rev : BOOL;   // Letoff Letoff A VFD Request Jog REV
   p20r15_request_over_speed : BOOL;   // Letoff Letoff A VFD Request Accumulator Over-Speed
        .CH0DATA   // Analog Input Splice Press Load Cell
        .CH1DATA   // Analog Input Tension Stand 1 Load Cell
        .CH2DATA   // Analog Input Winder Stand Load Cell
        .CH3DATA   // Analog Input Spare
        .CH4DATA   // Analog Input Letoff A Yardage
        .CH5DATA   // Analog Input Letoff B Yardage
        .CH6DATA   // Analog Input Winder A Yardage
        .CH7DATA   // Analog Input Winder B Yardage
   p20r15_request_position : BOOL;   // Letoff Letoff A VFD Request Accumulator Position Control
   p20r15_request_stop : BOOL := 1;   // Letoff Letoff A VFD Request Stop
   p20r15_request_tension : BOOL;   // Letoff Letoff A VFD Request Tension
   p20r15_request_thread_fwd : BOOL;
   p20r15_request_thread_rev : BOOL;
   p20r15_timer_fault : TIMER[10];   // Letoff Letoff A VFD Fault Timer
   p20r15_timer_warning : TIMER[5];   // Letoff Letoff A VFD Warning Dwell Timer
   p20r15_zero_speed : BOOL := 1;   // Letoff Letoff A VFD At Zero Speed
   p20r16 : routine := (comment := -536870793);   // Letoff Letoff B VFD
        .FAULT.0   // Letoff Letoff B VFD Drive Faulted
        .FAULT.2   // Letoff Letoff B VFD Drive Not Ready
        .FAULT.3   // Letoff Letoff B VFD Drive Not in Remote Mode
        .FAULT.4   // Letoff Letoff B VFD Motor Temperature
        .FAULT.5   // Letoff Letoff B Brake Temperature
        .WARNING   // Letoff Letoff B VFD
        .WARNING.0   // Letoff Letoff B VFD Warning
        .UNACK_FAULT   // Letoff Letoff B VFD Unacknowledged Faults Exists
        .UNACK_WARNING   // Letoff Letoff B VFD Unacknowledged Warning Exists
   p20r16_loa_accel_decel_ramp : SYS_ACC_DEC_RAMP := (IN_param_master_accel_rate := 2.0, IN_param_master_decel_rate := 20.0, IN_last_scan_s := 0.034016);   // Letoff Letoff B VFD Accel/Decel Ramp
   p20r16_lob_accel : REAL := 2.0;   // Letoff Letoff B VFD Accel Rate
   p20r16_lob_decel : REAL := 20.0;   // Letoff Letoff B VFD Decel Rate
   p20r16_lob_on : BOOL;   // Letoff Letoff B On
   p20r16_lob_selected_speed : REAL;   // Letoff Letoff B VFD Selected Speed
   p20r16_permissive_run : BOOL := 1;   // Letoff Letoff B VFD Permissive Run
   p20r16_request_jog_fwd : BOOL;   // Letoff Letoff B VFD Request Jog FWD
   p20r16_request_jog_rev : BOOL;   // Letoff Letoff B VFD Request Jog REV
   p20r16_request_over_speed : BOOL;   // Letoff Letoff B VFD Request Over Speed
   p20r16_request_position : BOOL;   // Letoff Letoff B VFD Request Position
   p20r16_request_stop : BOOL := 1;   // Letoff Letoff B VFD Request Stop
   p20r16_request_tension : BOOL;   // Letoff Letoff B VFD Request Tension
   p20r16_request_thread_fwd : BOOL;
   p20r16_request_thread_rev : BOOL;
   p20r16_timer_fault : TIMER[10];   // Letoff Letoff B VFD Fault Dwell Timer
   p20r16_timer_warning : TIMER[4];   // Letoff Letoff B VFD Warning Dwell Timer
   p20r16_zero_speed : BOOL := 1;   // Letoff Letoff B VFD Zero Speed
   p20r17 : routine := (comment := -1073741777);   // Letoff Letoff Diameter Calc
        .UNACK_FAULT   // Letoff Letoff Diameter Calc Unacknowledged Faults Exists
        .UNACK_WARNING   // Letoff Letoff Diameter Calc Unacknowledged Warning Exists
   p20r17_ave_control : CONTROL := (LEN := 19);   // Letoff Letoff Diameter Calc Average Control
   p20r17_diameter_clac_active : BOOL;   // Letoff Letoff Diameter Calc Active
   p20r17_letoff_avg_diam_inch : REAL := 26.150066;   // Letoff Letoff Diameter Calc Average Diameter [in]
   p20r17_letoff_diam_avg_stack : REAL[20] := ([0] := 26.174625, [1] := 26.174625, [2] := 26.143517, [3] := 26.174625, [4] := 26.143517, [5] := 26.143517, [6] := 26.143517, [7] := 26.174625, [8] := 26.174625, [9] := 26.143517, [10] := 26.143517, [11] := 26.112404, [12] := 26.174625, [13] := 26.143517, [14] := 26.112404, [15] := 26.143517, [16] := 26.174625, [17] := 26.112404, [18] := 26.112404);   // Letoff Letoff Diameter Calc Average Stack
   p20r17_stack_ctrl : CONTROL := (LEN := 20, POS := 19);   // Letoff Letoff Diameter Calc Stack Control
   p20r17_timer : TIMER[5] := ([0].PRE := 100, [1].PRE := 50);   // Letoff Letoff Diameter Calc Timer
   p20r17_timer_fault : TIMER[5];   // Letoff Letoff Diameter Calc Fault Dwell Timer
   p20r17_timer_warning : TIMER[5];   // Letoff Letoff Diameter Calc Warning Dwell Timer
   p20r17_winder_a_unload : REAL := 26.143517;   // Letoff Letoff Diameter Calc Temp Unload
   p20r18 : routine := (comment := -1073741321, state := 3);   // Letoff Letoff Turret VFD
        .FAULT.0   // Letoff Letoff Turret VFD Drive Faulted
        .FAULT.2   // Letoff Letoff Turret VFD Drive Not Ready
        .FAULT.3   // Letoff Letoff Turret VFD Drive Not in Remote Mode
        .FAULT.5   // Letoff Letoff Turret Motor Temperature
        .WARNING   // Letoff Letoff Turret VFD
        .WARNING.0   // Letoff Letoff Turret VFD Warning
        .WARNING.1   // Letoff Letoff Turret VFD Index Not Complete
        .WARNING.2   // Letoff Letoff Turret VFD No Letoff Selected
        .UNACK_FAULT   // Letoff Letoff Turret VFD Unacknowledged Faults Exists
        .UNACK_WARNING   // Letoff Letoff Turret VFD Unacknowledged Warning Exists
        .STATE.0   // Letoff Letoff Turret One Step Per Scan
        .STATE.1   // Letoff Letoff Turret Step 1: Idle
        .STATE.2   // Letoff Turret Step 2: Start Index Direction
        .STATE.3   // Letoff Letoff Turret Step 3: Index Active
        .STATE.4   // Letoff Letoff Turret Step 4: Prox Positive Transition
        .STATE.5   // Letoff Letoff Turret Step 5: Drive Stop
        .STATE.6   // Letoff Letoff Turret Step 6: Drive Slow Index Reverse Direction
        .STATE.7   // Letoff Letoff Turret Step 7:Stop Drive
        .STATE.8   // Letoff Letoff Turret Step 8: Index Complete
        .STATE.9   // Letoff Letoff Turret Step 9: Start Drive Forward
        .STATE.10   // Letoff Letoff Turret Step 10: Index Complete
   p20r18_acc_dec_ramp : SYS_ACC_DEC_RAMP := (IN_param_master_accel_rate := 8.0, IN_param_master_decel_rate := 8.0, IN_last_scan_s := 0.033844);   // Letoff Letoff Turret VFD Acel Decel Ramp
   p20r18_accel_rate : REAL := 8.0;
   p20r18_decel_rate : REAL := 8.0;
   p20r18_index_complete : BOOL := 1;   // Letoff Letoff Turret VFD Index Complete
   p20r18_index_move_timer : TIMER := (PRE := 7066);   // Letoff Letoff Turret VFD Move Timer
   p20r18_index_time : DINT := 7066;   // Letoff Letoff Turret Index Time
   p20r18_index_time_offset : DINT := 1250;   // Letoff Letoff Turret VFD Index Time Offset (Accel/Decel Rate Difference)
   p20r18_index_timer : TIMER := (PRE := 999999);   // Letoff Letoff Turret Index Timer
   p20r18_pb_index_fwd : BOOL;   // Letoff Letoff Turret VFD PB: Index FWD
   p20r18_pb_index_rev : BOOL;   // Letoff Letoff Turret VFD PB: Index REV
   p20r18_permissive : BOOL;   // Letoff Letoff Turret VFD Permissive
   p20r18_request_index_fwd : BOOL;   // Letoff Letoff Turret Request Index Forward
   p20r18_request_index_rev : BOOL;   // Letoff Letoff Turret Request Index Reverse
   p20r18_selected_speed : REAL;   // Letoff Letoff Turret VFD Selected Speed
   p20r18_timer_fault : TIMER[10] := ([3].PRE := 1000);   // Letoff Letoff Turret Fault Dwell Timer
   p20r18_timer_warning : TIMER[4] := ([1].PRE := 2000, [2].PRE := 2000);   // Letoff Letoff Turret VFD Warning Dwell Timer
   p20r18_zero_speed : BOOL := 1;   // Letoff Letoff Turret VFD At Zero Speed
   p21_ai_splice_platen_temp : REAL := 73.9;   // Splice Press Analog Input Platen Temperature
   p21_ao_splice_platen_temp_cv : REAL;   // Splice Press Analog Output Platen Temp Command Value
   p21_di_close_exit_clamp : BOOL;   // Splice Press Digital Input Close Exit Clamp
   p21_di_close_inlet_clamp : BOOL;   // Splice Press Digital Input Close Inlet Clamp
   p21_di_open_splice_platen : BOOL;   // Splice Press Digital Input Open Platen
   p21_di_platen_hi_temp_ok : BOOL := 1;   // Splice Press Digital Input Platen High Temperature Ok
   p21_di_platen_not_closed : BOOL := 1;   // Splice Press Digital Input Platen Not Closed
   p21_di_splice_2_hand_close : BOOL;   // Splice Press Digital Input Two Hand Switch Close Splicer
   p21_di_tc_bo : BOOL;   // Splice Press Digital Input Splice Platen Thermocouple Failure
   p21_dint_to_hmi : DINT[16] := ([10] := 2);   // Splice Press
        [0].0   // Splice Press Dint to HMI PI: Inlet Clamp Closed
        [0].1   // Splice Press Dint to HMI PI: Splice Press Closed
        [0].2   // Splice Press Dint to HMI PI: Exit Clamp Closed
        [0].3   // Splice Press Dint to HMI PI: Heater On
        [1]   // Splice Press Status
        [2]   // Splice Press Alarms
        [2].0   // Splice Press Alarms A00: Hardware High Limit
        [2].1   // Splice Press Alarms A01: Thermocouple Failure
        [2].2   // Splice Press Alarms A02
        [2].3   // Splice Press Alarms A03
        [2].4   // Splice Press Alarms A04
        [2].5   // Splice Press Alarms A05
        [2].6   // Splice Press Alarms A06
        [2].7   // Splice Press Alarms A07
        [2].8   // Splice Press Alarms A08
        [2].9   // Splice Press Alarms A09
        [2].10   // Splice Press Alarms A10
        [2].11   // Splice Press Alarms A11
        [2].12   // Splice Press Alarms A12
        [2].13   // Splice Press Alarms A13
        [2].14   // Splice Press Alarms A14
        [2].15   // Splice Press Alarms A15
        [2].16   // Splice Press Alarms A16
        [2].17   // Splice Press Alarms A17
        [2].18   // Splice Press Alarms A18
        [2].19   // Splice Press Alarms A19
        [2].20   // Splice Press Alarms A20
        [2].21   // Splice Press Alarms A21
        [2].22   // Splice Press Alarms A22
        [2].23   // Splice Press Alarms A23
        [2].24   // Splice Press Alarms A24
        [2].25   // Splice Press Alarms A25
        [2].26   // Splice Press Alarms A26
        [2].27   // Splice Press Alarms A27
        [2].28   // Splice Press Alarms A28
        [2].29   // Splice Press Alarms A29
        [2].30   // Splice Press Alarms A30
        [2].31   // Splice Press Alarms A31
        [4].0   // Splice Press Warning W00: Platen Heater Not On
        [4].1   // Splice Press Warning W01:
        [4].2   // Splice Press Warning W02:
        [4].3   // Splice Press Warning W03:
        [4].4   // Splice Press Warning W04:
        [4].5   // Splice Press Warning W05:
        [4].6   // Splice Press Warning W06:
        [4].7   // Splice Press Warning W07:
        [4].8   // Splice Press Warning W08:
        [4].9   // Splice Press Warning W09:
        [4].10   // Splice Press Warning W10:
        [4].11   // Splice Press Warning W11:
        [4].12   // Splice Press Warning W12:
        [4].13   // Splice Press Warning W13:
        [4].14   // Splice Press Warning W14:
        [4].15   // Splice Press Warning W15:
        [4].16   // Splice Press Warning W16:
        [4].17   // Splice Press Warning W17:
        [4].18   // Splice Press Warning W18:
        [4].19   // Splice Press Warning W19:
        [4].20   // Splice Press Warning W20:
        [4].21   // Splice Press Warning W21:
        [4].22   // Splice Press Warning W22:
        [4].23   // Splice Press Warning W23:
        [4].24   // Splice Press Warning W24:
        [4].25   // Splice Press Warning W25:
        [4].26   // Splice Press Warning W26:
        [4].27   // Splice Press Warning W27:
        [4].28   // Splice Press Warning W28:
        [4].29   // Splice Press Warning W29:
        [4].30   // Splice Press Warning W30:
        [4].31   // Splice Press Warning W31:
   p21_do_close_exit_clamp_sv : BOOL;   // Splice Press Digital Output Close Exit Clamp
   p21_do_close_inlet_clamp_sv : BOOL;   // Splice Press Digital Output Close Inlet Clamp
   p21_do_close_platen_sv : BOOL;   // Splice Press Digital Output Close Splicer Press
   p21_do_enable_platen_heater : BOOL;   // Splice Press Digital Output Enable Platen Heater
   p21_pid_splice_press_temp : PID := (CTL := -2077195136, EN := 1, SWM := 1, NOBC := 1, NOZC := 1, INI := 1, DVNA := 1, PVHA := 1, KP := 30.0, BIAS := 30.0, MAXS := 1000.0, MAXO := 100.0, UPD := 0.01, PV := 74.1, ERR := -74.1, MAXI := 1000.0, MAXCV := 100.0, MAXTIE := 100.0, DATA[1] := -118.56, DATA[2] := 74.1, DATA[3] := -74.1, DATA[5] := 0.1, DATA[6] := 1.0, DATA[7] := 0.16, DATA[8] := 30.0, DATA[11] := 30.0, DATA[15] := 1.0, DATA[16] := 1.0);   // Splice Press Temperature Control PID
   p21_real_to_hmi : REAL[112] := ([0] := 74.1, [1] := 55.0);   // Splice Press Real to HMI
   p21_splice_press_temp_out : SYS_SCP := (Input_Max := 100.0, Output_Max := 32767.0, Output := -0.001953125);   // Splice Press Analog Ouputs Platen Heater
   p21_splice_temp_in_max : REAL := 100.0;
   p21_splice_temp_in_min : REAL;
   p21_splice_temp_out_max : REAL := 32767.0;
   p21_splice_temp_out_min : REAL;
   P21r01 : routine := (comment := 7);
   p21r02 : routine := (comment := -1073741761);   // Splice Press Misc Control
        .UNACK_FAULT   // Splice Press Misc Control Unacknowledged Fault Exists
        .UNACK_WARNING   // Splice Press Misc Control Unacknowledged Warning Exists
   p21r02_fault_exists : BOOL;
   p21r02_timer_fault : TIMER[4];   // Splice Press Misc Control Fault Delay
   p21r02_timer_warning : TIMER[4];   // Splice Press Misc Control Warning Delay
   p21r02_unack_fault : BOOL;   // Splice Press Misc Control Unacknowledged Fault Exists
   p21r02_unack_warning : BOOL;   // Splice Press Misc Control Unacknowledged Warning Exists
   p21r02_warning_exists : BOOL;
   p21r03 : routine := (comment := -1073741761);   // Splice Press Inputs
        .UNACK_FAULT   // Splice Press input Unacknowledged Fault Exists
        .UNACK_WARNING   // Splice Press Input Unacknowledged Warning Exists
   p21r03_timer_fault : TIMER[4];   // Splice Press Input Fault Dwell Timer
   p21r03_timer_warning : TIMER[4];   // Splice Press Input Warning Dwell Timer
   p21r04 : routine := (comment := -1073741761);   // Splice Press Outputs
        .UNACK_FAULT   // Splice Press Output Unacknowledged Fault Exists
        .UNACK_WARNING   // Splice Press Output Unacknowledged Warning Exists
   p21r04_timer_fault : TIMER[4];   // Splice Press Outputs Fault Delay
   p21r04_timer_warning : TIMER[4];   // Splice Press Outputs Warning Delay
   p21r05 : routine := (comment := -1073741761);   // Splice Press Dint to HMI
        .UNACK_FAULT   // Splice Press Dint to HMI Unacknowledged Fault Exists
        .UNACK_WARNING   // Splice Press Dint to HMI Unacknowledged Warning Exists
   p21r05_timer_fault : TIMER[4];   // Splice Press Dint to HMI Fault Delay
   p21r05_timer_warning : TIMER[4];   // Splice Press Dint to HMI Warning Delay
   p21r06 : routine := (comment := -1073741796);   // Splice Press Real to HMI
        .UNACK_FAULT   // Splice Press Real to HMI Unacknowledged Fault Exists
        .UNACK_WARNING   // Splice Press Real to HMI Unacknowledged Warning Exists
   p21r06_timer_fault : TIMER[4];   // Splice Press Real to HMI Fault Delay
   p21r06_timer_warning : TIMER[4];   // Splice Press Real to HMI Warning Delay
   p21r07 : routine := (comment := -1073741761);   // Splice Press Alarms
        .UNACK_FAULT   // Splice Press Alarms Unacknowledged Fault Exists
        .UNACK_WARNING   // Splice Press Alarms Unacknowledged Warning Exists
   p21r07_timer_fault : TIMER[4];   // Splice Press Alarms Fault Delay
   p21r07_timer_warning : TIMER[4];   // Splice Press Alarms Warning Delay
   p21r08 : routine := (comment := -1073741761);   // Splice Press Warnings
        .UNACK_FAULT   // Splice Press Warnings Unacknowledged Fault Exists
        .UNACK_WARNING   // Splice Press Warnings Unacknowledged Warning Exists
   p21r08_timer_fault : TIMER[4];   // Splice Press Warnings Fault Delay
   p21r08_timer_warning : TIMER[4];   // Splice Press Warnings Warning Delay
   p21r09 : routine := (comment := -1073741761);   // Splice Press Modes
        .UNACK_FAULT   // Splice Press Modes Unacknowledged Fault Exists
        .UNACK_WARNING   // Splice Press Modes Unacknowledged Warning Exists
   p21r09_timer_fault : TIMER[4];   // Splice Press Modes Fault Delay
   p21r09_timer_warning : TIMER[4];   // Splice Press Modes Warning Delay
   p21r10 : routine := (comment := -1073741761);   // Splice Press Sequence
        .FAULT.0   // Splice Press Sequence Sequence Not Complete
        .UNACK_FAULT   // Splice Press Sequence Unacknowledged Fault Exists
        .UNACK_WARNING   // Splice Press Sequence Unacknowledged Warning Exists
   p21r10_index_kd : REAL;
   p21r10_index_ki : REAL := 0.1;
   p21r10_index_kp : REAL := 1.0;
   p21r10_permissive_run : BOOL := 1;   // Splice Press Sequence Permissive Run
   p21r10_remaining_cure_time : DINT := 55000;
   p21r10_remaining_cure_time_sec : REAL := 55.0;   // Splice Press Sequence Remaining Cure Timer [Sec]
   p21r10_splice_press_1 : SYS_ENC := (IN_State := 5, OUT_Status := 2);   // Splice Press Sequence Encoder
   p21r10_state : DINT := 5;   // Splice Press Sequence State
        .0   // Splice Press Sequence State 0 One Step Per Scan
        .1   // Splice Press Sequence State 1 Idle
        .2   // Splice Press Sequence State 2 Enable Sequence
        .3   // Splice Press Sequence State 3 Close Exit Clamp
        .4   // Splice Press Sequence State 4 Close Inlet Clamp
        .5   // Splice Press Sequence State 5 Closing Platen
        .6   // Splice Press Sequence State 6 Cure in Progress
        .7   // Splice Press Sequence State 7 Cure Done
        .8   // Splice Press Sequence State 8 Platen Open
        .9   // Splice Press Sequence State 9 Inlet Clamp Open
        .10   // Splice Press Sequence State 10 Exit Clamp Open
        .11   // Splice Press Sequence State 11 Complete
   p21r10_status : DINT := 2;   // Splice Press Sequence Status
   p21r10_timer_exit_open_delay : TIMER;   // Splice Press Sequence Exit Open Delay
   p21r10_timer_fault : TIMER[4];   // Splice Press Sequence Fault Delay
   p21r10_timer_inlet_open_delay : TIMER;   // Splice Press Sequence Inlet Open Delay
   p21r10_timer_platen_open_delay : TIMER;   // Splice Press Sequence Platen Open Delay
   p21r10_timer_press_cure : TIMER := (PRE := 55000);   // Splice Press Sequence Press Cure Dwell
   p21r10_timer_warning : TIMER[4];   // Splice Press Sequence Warning Delay
   p21r11_index_kd : REAL;
   p21r11_index_ki : REAL := 0.1;
   p21r11_index_kp : REAL := 1.2;
   p21r11_run_kd : REAL;
   p21r11_run_ki : REAL := 0.8;
   p21r11_run_kp : REAL := 1.0;
   p21r16 : routine := (comment := -1073741697, oneshot := 1024);   // Splice Press Temperature Control
        .FAULT.0   // Splice Press Temperature Control Hardware High Limit
        .FAULT.1   // Splice Press Temperature Control Thermocouple Failure
        .WARNING.0   // Splice Press Temperature Control Platen Heater Not On Warning
        .UNACK_FAULT   // Splice Press Temperature Control Unacknowledged Fault Exists
        .UNACK_WARNING   // Splice Press Temperature Control Unacknowledged Warning Exists
   p21r16_pb_heater_off : BOOL;   // Splice Press Temperature Control PB: Heater Off
   p21r16_pb_heater_on : BOOL;   // Splice Press Temperature Control PB: Heater On
   p21r16_permissive_run : BOOL := 1;   // Splice Press Temperature Control Permissive Run
   p21r16_pid_temp_cv : REAL;   // Splice Press Temperature Control PID Control Variable
   p21r16_pid_temp_pv : REAL := 73.9;   // Splice Press Temperature Control PID Process Variable
   p21r16_pid_timer : TIMER := (ACC := 32, EN := 1, DN := 1);   // Splice Press Temperature Control PID Enable Timer
   p21r16_request_heat : BOOL;   // Splice Press Temperature Control Request Heat
   p21r16_timer_fault : TIMER[16] := ([2].PRE := 2000);   // Splice Press Temperature Control Fault Delay
   p21r16_timer_warning : TIMER[16];   // Splice Press Temperature Control Warning Delay
   p22_ai_amps : REAL;   // Tension Stand 1 Analog Input Tension Stand 1 Motor Current
   p22_ai_hz : REAL;   // Tension Stand 1 Analog Input Tension Stand 1 Motor Hertz
   p22_ai_speed : REAL;
   p22_ai_torque : REAL;
   p22_ai_ts1_lc : REAL := 57.124866;   // Tension Stand 1 Analog Input Loadcell
   p22_ao_selected_speed : REAL;   // Tension Stand 1 VFD Selected Speed
   p22_ao_torque : REAL := 300.0;
   p22_ao_vfd : REAL;
   p22_control_word : INT := 2#0000_0100_0000_0111;
   p22_di_brake : BOOL := 1;   // Tension Stand 1 Digital Input Brake Temperature OK
   p22_di_close_nip_roll : BOOL;   // Tension Stand 1 Digital Input SS: Close Nip Roll
   p22_di_jog : BOOL;   // Tension Stand 1 Digital Input SS: Jog
   p22_di_jog_fwd : BOOL;   // Tension Stand 1 Digital Input PB: Jog Forward
   p22_di_jog_rev : BOOL;   // Tension Stand 1 Digital Input PB: Jog Reverse
   p22_di_open_nip_roll : BOOL := 1;   // Tension Stand 1 Digital Input SS: Open Nip Roll
   p22_di_run : BOOL := 1;   // Tension Stand 1 Digital Input SS: Run
   p22_di_therm : BOOL := 1;   // Tension Stand 1 Digital Input Motor Temperature OK
   p22_dint_to_hmi : DINT[16] := ([0] := 4, [1] := 4915, [7] := 2);   // Tension Stand 1 Dint to HMI
        [0].0   // Tension Stand 1 Dint to HMI Nip Closed
        [1].0   // Tension Stand 1 Dint to HMI VFD Faulted
        [1].1   // Tension Stand 1 Dint to HMI VFD Warning
        [1].2   // Tension Stand 1 Dint to HMI VFD Running Forward
        [1].3   // Tension Stand 1 Dint to HMI VFD Running Reverse
        [1].4   // Tension Stand 1 Dint to HMI VFD Ready
        [1].5   // Tension Stand 1 Dint to HMI VFD Control From Net
        [1].6   // Tension Stand 1 Dint to HMI VFD Reference From Net
        [1].7   // Tension Stand 1 Dint to HMI VFD at Reference
        [2].0   // Tension Stand 1 Alarms A00: VFD Faulted
        [2].1   // Tension Stand 1 Alarms A01: VFD Motor Brake Failure
        [2].2   // Tension Stand 1 Alarms A02: VFD Not Ready
        [2].3   // Tension Stand 1 Alarms A03: VFD Not in Network Mode
        [2].4   // Tension Stand 1 Alarms A04: VFD Motor Temperature
        [2].5   // Tension Stand 1 Alarms A05: VFD Motor Brake Temperature
        [2].6   // Tension Stand 1 Alarms A06:
        [2].7   // Tension Stand 1 Alarms A07:
        [2].8   // Tension Stand 1 Alarms A08:
        [2].9   // Tension Stand 1 Alarms A09:
        [2].10   // Tension Stand 1 Alarms A10:
        [2].11   // Tension Stand 1 Alarms A11:
        [2].12   // Tension Stand 1 Alarms A12:
        [2].13   // Tension Stand 1 Alarms A13:
        [2].14   // Tension Stand 1 Alarms A14:
        [2].15   // Tension Stand 1 Alarms A15:
        [2].16   // Tension Stand 1 Alarms A16:
        [2].17   // Tension Stand 1 Alarms A17:
        [2].18   // Tension Stand 1 Alarms A18:
        [2].19   // Tension Stand 1 Alarms A19:
        [2].20   // Tension Stand 1 Alarms A20:
        [2].21   // Tension Stand 1 Alarms A21:
        [2].22   // Tension Stand 1 Alarms A22:
        [2].23   // Tension Stand 1 Alarms A23:
        [2].24   // Tension Stand 1 Alarms A24:
        [2].25   // Tension Stand 1 Alarms A25:
        [2].26   // Tension Stand 1 Alarms A26:
        [2].27   // Tension Stand 1 Alarms A27:
        [2].28   // Tension Stand 1 Alarms A28:
        [2].29   // Tension Stand 1 Alarms A29:
        [2].30   // Tension Stand 1 Alarms A30:
        [2].31   // Tension Stand 1 Alarms A31:
        [4].0   // Tension Stand 1 Warning W00: Tension Stand 1 VFD Warning
        [4].1   // Tension Stand 1 Warning W01:
        [4].2   // Tension Stand 1 Warning W02:
        [4].3   // Tension Stand 1 Warning W03:
        [4].4   // Tension Stand 1 Warning W04: Tension Stand 1 not in Run Mode
        [4].5   // Tension Stand 1 Warning W05
        [4].6   // Tension Stand 1 Warning W06:
        [4].7   // Tension Stand 1 Warning W07:
        [4].8   // Tension Stand 1 Warning W08
        [4].9   // Tension Stand 1 Warning W09
        [4].10   // Tension Stand 1 Warning W10
        [4].11   // Tension Stand 1 Warning W11
        [4].12   // Tension Stand 1 Warning W12
        [4].13   // Tension Stand 1 Warning W13
        [4].14   // Tension Stand 1 Warning W14
        [4].15   // Tension Stand 1 Warning W15
        [4].16   // Tension Stand 1 Warning W16
        [4].17   // Tension Stand 1 Warning W17
        [4].18   // Tension Stand 1 Warning W18
        [4].19   // Tension Stand 1 Warning W19
        [4].20   // Tension Stand 1 Warning W20
        [4].21   // Tension Stand 1 Warning W21
        [4].22   // Tension Stand 1 Warning W22
        [4].23   // Tension Stand 1 Warning W23
        [4].24   // Tension Stand 1 Warning W24
        [4].25   // Tension Stand 1 Warning W25
        [4].26   // Tension Stand 1 Warning W26
        [4].28   // Tension Stand 1 Warning W28
        [4].29   // Tension Stand 1 Warning W29
        [4].30   // Tension Stand 1 Warning W30
        [4].31   // Tension Stand 1 Warning W31
   p22_do_close_nip_roll : BOOL;   // Tension Stand 1 Digital Output Close Tension Stand 1 Nip Roll
   p22_param_ts1_jog_speed : REAL := 8.0;   // System Parameter Tension Stand 1 Jog Speed
   p22_real_to_hmi : REAL[112] := ([0] := 57.09026, [40] := 4.2, [41] := 2.0, [42] := 5.0);   // Tension Stand 1 Real to HMI
        [6]   // Tension Stand 1 Real to HMI VFD Hertz
        [7]   // Tension Stand 1 Real to HMI VFD Amps
        [8]   // Tension Stand 1 Real to HMI VFD Hertz
   p22_status_word : INT := 2#0001_0011_0011_0011;
   p22_ts1_acc_rate : REAL := 8.0;
   p22_ts1_decel_rate : REAL := 8.0;
   p22_ts1_gear_ratio : REAL := 54.76;
   p22_ts1_roll_diameter_ft : REAL := 0.5;
   p22_ts1_vfd : ABB_PROTOCOL_VFD := (STATUS_WORD := 4915, CONTROL_WORD := 1031, IN_DRIVE_PERMISSIVE := 1);
   p22_vfd_input_max : REAL := 2000.0;
   p22_vfd_input_min : REAL := -2000.0;
   p22_vfd_output_max : REAL := 20000.0;
   p22_vfd_output_min : REAL := -20000.0;
   p22r01 : routine := (comment := 7);   // Tension Stand 1 Main
   p22r02 : routine := (comment := -1073741761);   // Tension Stand 1 Misc Control
        .FAULT.0   // Tension Stand 1 Misc Control Oil Pressure Failure
        .UNACK_FAULT   // Tension Stand 1 Misc Control Unaknowledged Fault Exists
        .UNACK_WARNING   // Tension Stand 1 Misc Control Unaknowledged Warning Exists
   p22r02_fault_exists : BOOL;
   p22r02_nip_open : BOOL := 1;
   p22r02_nip_open_dwell : TIMER := (PRE := 2000, ACC := 2011, EN := 1, DN := 1);
   p22r02_request_system_run : BOOL;   // Tension Stand 1 Misc Control Request System Run
   p22r02_tension_dev_max : REAL := 56.0;   // Winder A VFD
        .DATA[0]   // Output Winder A VFD Control Word
        .DATA[0].0   // Output Winder A VFD Run Forward
        .DATA[0].1   // Output Winder A VFD Run Reverse
        .DATA[0].2   // Output Winder A VFD Fault Reset
        .DATA[0].5   // Output Winder A VFD Net Control
        .DATA[0].6   // Output Winder A VFD Net Reference
        .DATA[1]   // Output Winder A VFD Speed Command
   p22r02_tension_dev_min : REAL := 44.0;   // Tension Stand 1 VFD
        .DATA[0]   // Output Tension Stand 1 VFD Control Word
        .DATA[0].0   // Output Tension Stand 1 VFD Run Forward
        .DATA[0].1   // Output Tension Stand 1 VFD Run Reverse
        .DATA[0].2   // Output Tension Stand 1 VFD Fault Reset
        .DATA[0].5   // Output Tension Stand 1 VFD Net Control
        .DATA[0].6   // Output Tension Stand 1 VFD Net Reference
        .DATA[1]   // Output Tension Stand 1 VFD Speed Command
   p22r02_timer_fault : TIMER[4];   // Tension Stand 1 Misc Control Fault Delay
   p22r02_timer_warning : TIMER[4];   // Tension Stand 1 Misc Control Warning Delay
   p22r02_unack_fault : BOOL;   // Impreg Pickup Roll Misc Control Unacknowledged Fault Exists
   p22r02_unack_warning : BOOL;   // Impreg Pickup Roll Misc Control Unacknowledged Warning Exists
   p22r02_warning_exists : BOOL;
   p22r03 : routine := (comment := -1073741761);   // Tension Stand 1 Input
        .UNACK_FAULT   // Tension Stand 1 Input Unaknowledged Fault Exists
        .UNACK_WARNING   // Tension Stand 1 Input Unaknowledged Warning Exists
   p22r03_ave_tq : REAL;
   p22r03_hz : SYS_SCP := (Input_Max := 2000.0, Output_Max := 60.0);   // Tension Stand 1 Analog Inputs SCP Hz
   p22r03_lc_input_max : REAL := 10000.0;
   p22r03_lc_input_min : REAL;
   p22r03_lc_output_max : REAL := 250.0;
   p22r03_lc_output_min : REAL;
   p22r03_lc_scp : SYS_SCP := (Input := 2284.0132, Input_Max := 10000.0, Output_Max := 250.0, Output := 57.10033);   // Tension Stand 1 Analog Input Load Cell Scaling
   p22r03_sample_timer : TIMER := (PRE := 200, ACC := 132, EN := 1, TT := 1);
   p22r03_scaled_vfd_in : REAL;
   p22r03_timer_fault : TIMER[4];   // Tension Stand 1 Input Fault Delay
   p22r03_timer_warning : TIMER[4];   // Tension Stand 1 Input Warning Delay
   p22r03_tq_ave_ctrl : CONTROL := (LEN := 19);
   p22r03_tq_buffer : REAL[20];
   p22r03_tq_fifo : CONTROL := (LEN := 20, POS := 20, DN := 1);
   p22R03_ts1_vfd_rpm_to_speed : SYS_RPM_TO_SPEED := (IN_gear_ratio := 54.76, IN_roll_diameter := 0.5);   // Tension Stand 1 Analog Input VFD RPM to Roll Surface Speed
   p22r03_unload : DINT;
   p22r03_vfd_in_scaling : SYS_SCP := (Input_Min := -20000.0, Input_Max := 20000.0, Output_Min := -2000.0, Output_Max := 2000.0);
   p22r03_vfd_input_max : REAL := 20000.0;
   p22r03_vfd_input_min : REAL := -20000.0;
   p22r03_vfd_out_scaling : SYS_SCP := (Input_Min := -2000.0, Input_Max := 2000.0, Output_Min := -20000.0, Output_Max := 20000.0);
   p22r03_vfd_output_max : REAL := 2000.0;
   p22r03_vfd_output_min : REAL := -2000.0;
   p22r04 : routine := (comment := -1073741761);   // Tension Stand 1 Output
        .UNACK_FAULT   // Tension Stand 1 Output Unaknowledged Fault Exists
        .UNACK_WARNING   // Tension Stand 1 Output Unaknowledged Warning Exists
   p22r04_speed_to_vfd_1 : SYS_SPEED_TO_VFD := (IN_gear_ratio := 54.76, IN_roll_diameter := 0.5);   // Tension Stand 1 Analog Output Speed to VFD
   p22r04_timer_fault : TIMER[4];   // Tension Stand 1 Output Fault Delay
   p22r04_timer_warning : TIMER[4];   // Tension Stand 1 Output Warning Delay
   p22r05 : routine := (comment := -1073741761);   // Tension Stand 1 Dint to HMI
        .UNACK_FAULT   // Tension Stand 1 Dint to HMI Unaknowledged Fault Exists
        .UNACK_WARNING   // Tension Stand 1 Dint to HMI Unaknowledged Warning Exists
   p22r05_timer_fault : TIMER[4];   // Tension Stand 1 Dint to HMI Fault Delay
   p22r05_timer_warning : TIMER[4];   // Tension Stand 1 Dint to HMI Warning Delay
   p22r06 : routine := (comment := -1073741572);   // Tension Stand 1 Real to HMI
        .UNACK_FAULT   // Tension Stand 1 Real to HMI Unaknowledged Fault Exists
        .UNACK_WARNING   // Tension Stand 1 Real to HMI Unaknowledged Warning Exists
   p22r06_ave_lc : REAL := 57.12177;
   p22r06_lc_buffer : REAL[20] := ([0] := 57.08561, [1] := 57.110146, [2] := 57.110146, [3] := 57.105236, [4] := 57.095425, [5] := 57.095425, [6] := 57.095425, [7] := 57.10033, [8] := 57.0807, [9] := 57.0807, [10] := 57.105236, [11] := 57.095425, [12] := 57.090515, [13] := 57.095425, [14] := 57.090515, [15] := 57.095425, [16] := 57.08561, [17] := 57.095425, [18] := 57.095425, [19] := 57.090515);
   p22r06_lc_ctrl : CONTROL := (LEN := 20, POS := 20, DN := 1);
   p22r06_sample_timer : TIMER;
   p22r06_timer_fault : TIMER[4];   // Tension Stand 1 Real to HMI Fault Delay
   p22r06_timer_warning : TIMER[4];   // Tension Stand 1 Real to HMI Warning Delay
   p22r06_unload : DINT := 57;
   p22r07 : routine := (comment := -1073741761);   // Tension Stand 1 Alarms
        .UNACK_FAULT   // Tension Stand 1 Alarms Unaknowledged Fault Exists
        .UNACK_WARNING   // Tension Stand 1 Alarms Unaknowledged Warning Exists
   p22r07_timer_fault : TIMER[4];   // Tension Stand 1 Alarms Fault Delay
   p22r07_timer_warning : TIMER[4];   // Tension Stand 1 Alarms Warning Delay
   p22r08 : routine := (comment := -1073741761);   // Tension Stand 1 Warnings
        .UNACK_FAULT   // Tension Stand 1 Warnings Unaknowledged Fault Exists
        .UNACK_WARNING   // Tension Stand 1 Warnings Unaknowledged Warning Exists
   p22r08_timer_fault : TIMER[4];   // Tension Stand 1 Warnings Fault Delay
   p22r08_timer_warning : TIMER[4];   // Tension Stand 1 Warnings Warning Delay
   p22r09 : routine := (comment := -1073741761, fault := 1, fault_ack := 1);   // Tension Stand 1 Modes
        .WARNING.0   // Tension Stand 1 Modes Not in Run Mode
        .WARNING.1   // Tension Stand 1 Modes Tension Stand in Thread Mode
        .UNACK_FAULT   // Tension Stand 1 Modes Unaknowledged Fault Exists
        .UNACK_WARNING   // Tension Stand 1 Modes Unaknowledged Warning Exists
   p22r09_mode_jog : BOOL;   // Tension Stand 1 Modes Jog Mode
   p22r09_mode_run : BOOL := 1;   // Tension Stand 1 Modes Run Mode
   p22r09_mode_thread : BOOL;   // Tension Stand 1 Modes Thread Mode
   p22r09_pb_jog_fwd : BOOL;   // Tension Stand 1 Modes PB: Jog Forward
   p22r09_pb_jog_rev : BOOL;   // Tension Stand 1 Modes PB: Jog Reverse
   p22r09_timer_fault : TIMER[4];   // Tension Stand 1 Modes Fault Delay
   p22r09_timer_warning : TIMER[4];   // Tension Stand 1 Modes Warning Delay
   p22r10 : routine := (comment := -1073741761);   // Tension Stand 1 Speed Tension
        .UNACK_FAULT   // Tension Stand 1 Speed Tension Unaknowledged Fault Exists
        .UNACK_WARNING   // Tension Stand 1 Speed Tension Unaknowledged Warning Exists
   p22r10_calc_speed_offset : REAL;
   p22r10_param_psn_gain : REAL := 20.0;   // Tension Stand 1 Parameter Position Gain
   p22r10_pid_out : REAL := 50.0;
   p22r10_pid_psn : PID := (CTL := -1004501888, EN := 1, CT := 1, SWM := 1, NOBC := 1, INI := 1, DVNA := 1, PVHA := 1, SP := 50.0, KP := 4.2, KI := 2.0, KD := 5.0, BIAS := 1.0, MAXS := 500.0, SO := 50.0, MAXO := 100.0, UPD := 0.01, PV := 57.095425, ERR := -7.0954247, OUT := 50.0, MAXI := 500.0, MAXCV := 100.0, MAXTIE := 100.0, DATA[0] := 54.926666, DATA[1] := -182.73886, DATA[2] := 57.095425, DATA[3] := -7.0954247, DATA[4] := 50.0, DATA[5] := 0.2, DATA[6] := 1.0, DATA[7] := 5.16, DATA[8] := 4.2, DATA[9] := 2.0, DATA[10] := 5.0, DATA[11] := 4.2, DATA[12] := 2.0, DATA[13] := 5.0, DATA[15] := 1.0, DATA[16] := 1.0);   // Tension Stand 1 Speed Tension PID Dancer Position
   p22r10_pid_psn_cv : REAL := 50.0;   // Tension Stand 1 Speed Tension PID Dancer Position Control Variable
   p22r10_pid_psn_pv : REAL := 57.11505;   // Tension Stand 1 Speed Tension PID Dancer Position Process Variable
   p22r10_selected_torque : REAL := 300.0;
   p22r10_speed_offset : REAL;   // Tension Stand 1 Speed tension Speed Offset from Base
   p22r10_stretch : REAL;
   p22r10_timer_fault : TIMER[4];   // Tension Stand 1 Speed Tension Fault Delay
   p22r10_timer_warning : TIMER[4];   // Tension Stand 1 Speed Tension Warning Delay
   p22r11 : routine := (comment := -1073741713);   // Tension Stand 1 VFD
        .FAULT.0   // Tension Stand 1 VFD Drive Fault
        .FAULT.2   // Tension Stand 1 VFD Not Ready
        .FAULT.3   // Tension Stand 1 VFD Not in Network Mode
        .FAULT.4   // Tension Stand 1 VFD Motor Temperature
        .FAULT.5   // Tension Stand 1 VFD Motor Brake Temperature
        .WARNING.0   // Tension Stand 1 VFD Drive Warning
        .UNACK_FAULT   // Tension Stand 1 VFD Unaknowledged Fault Exists
        .UNACK_WARNING   // Tension Stand 1 VFD Unaknowledged Warning Exists
   p22r11_acc_decel_ramp : SYS_ACC_DEC_RAMP := (IN_param_master_accel_rate := 8.0, IN_param_master_decel_rate := 8.0, IN_last_scan_s := 0.033136);   // Tension Stand 1 VFD Accel/Decel Ramp
   p22r11_permissive_jog : BOOL := 1;   // Tension Stand 1 VFD Permissive Run
   p22r11_request_jog_fwd : BOOL;   // Tension Stand 1 VFD Request Jog FWD
   p22r11_request_jog_rev : BOOL;   // Tension Stand 1 VFD Request Jog REV
   p22r11_request_line_jog : BOOL;   // Tension Stand 1 VFD Request Line Jog
   p22r11_request_line_run : BOOL;   // Tension Stant 1 VFD Request Line Run
   p22r11_request_start : BOOL;   // Tension Stand 1 VFD
        .DATA[0]   // Input Tension Stand 1 VFD Status Word
        .DATA[0].0   // Input Tension Stand 1 VFD Faulted
        .DATA[0].1   // Input Tension Stand 1 VFD Warning
        .DATA[0].2   // Input Tension Stand 1 VFD Running Forward
        .DATA[0].3   // Input Tension Stand 1 VFD Running Reverse
        .DATA[0].4   // Input Tension Stand 1 VFD Ready
        .DATA[0].5   // Input Tension Stand 1 VFD Control from Net
        .DATA[0].6   // Input Tension Stand 1 VFD Reference from Net
        .DATA[0].7   // Input Tension Stand 1 VFD At Reference
        .DATA[1]   // Input Tension Stand 1 VFD Speed
        .DATA[2]   // Input Tension Stand 1 VFD Amps
        .DATA[3]   // Input Tension Stand 1 VFD Max Hertz
        .DATA[4]   // Input Tension Stand 1 VFD Motor Nameplate Hertz
        .DATA[5]   // Input Tension Stand 1 VFD Motor Nameplate RPM
   p22r11_request_tension : BOOL;
   p22r11_request_thread_fwd : BOOL;   // Tension Stand 1 VFD Request Thread FWD
   p22r11_request_thread_rev : BOOL;   // Tension Stand 1 VFD Request Thread REV
   p22r11_selected_speed : REAL;   // Tension Stand 1 VFD Selected Speed
   p22r11_timer_fault : TIMER[10];   // Tension Stand 1 VFD Fault Timer
   p22r11_timer_warning : TIMER[5] := ([1].PRE := 10000, [2].PRE := 10000);   // Tension Stand 1 VFD Warning Timer
   p22r11_zero_speed : BOOL := 1;   // Tension Stand 1 VFD Zero Speed
   p23_ai_ds_gap_dint : DINT := 70;
   p23_ai_ds_masked_gap : REAL := 0.007;
   p23_ai_lfl : REAL := 1.7023346;   // Impreg Inputs LFL level
   p23_ai_metering_roll_amps : REAL;   // Impreg Analog Input Impreg Metering Roll Motor Current
   p23_ai_metering_roll_hz : REAL := 3.8146973e-06;   // Impreg Analog Input Impreg Metering Roll Motor Max Hz
   p23_ai_metering_roll_speed_fpm : REAL;   // Impreg Analog Input Impreg Roll Speed
   p23_ai_os_gap_dint : DINT := 75;
   p23_ai_os_masked_gap : REAL := 0.0075;
   p23_ai_prs : REAL := -0.00967899;   // Impreg Analog Inputs Impreg Enclosure Pressure
   p23_ai_servo_ds_position : REAL := 0.007;   // Impreg Servo Drive Side Actual Position
   p23_ai_servo_ds_torque : REAL := 6553.2;   // Impreg Servo Drive Side Actual Torque
   p23_ai_servo_ds_velocity : REAL;   // Impreg Servo Drive Side Velocity Feedback
   p23_ai_servo_os_position : REAL := 0.0075000003;   // Impreg Inputs Servo Operator Side Position
   p23_ai_servo_os_torque : REAL := 65534.0;   // Impreg Inputs Servo Operator Side Torque
   p23_ai_servo_os_velocity : REAL;   // Impreg Inputs Servo Operator Side Velocity
   p23_ai_supply_amps : REAL;   // Impreg Analog Inputs Supply Fan VFD Amps
   p23_ai_supply_hz : REAL := 60.0;   // Impreg Analog Inputs Supply Fan VFD Hz
   p23_ai_supply_rpm : REAL;   // Impreg Analog Inputs Supply Fan RPM
   p23_ao_selected_speed : REAL;   // Impreg Metering Roll VFD Selected Speed
   p23_ao_servo_ds_jog_vel_cmd : REAL := 0.005;   // Impreg Servo Drive Side Jog Velocity Command [in/sec]
   p23_ao_servo_ds_position_cmd : REAL := 0.032;   // Impreg Servo Drive Side Position Command
   p23_ao_servo_ds_velocity_cmd : REAL := 0.011;   // Impreg Servo Drive Side Velocity Command
   p23_ao_servo_ds_zero_offset : REAL := 0.036;   // Impreg Analog Outputs Drive Side Servo Position Offset
   p23_ao_servo_os_jog_vel_cmd : REAL := -0.005;   // Impreg Servo Operator Side Jog Velocity Command [in/sec]
   p23_ao_servo_os_position_cmd : REAL := 0.033;   // Impreg Servo Operator Side Position Command
   p23_ao_servo_os_velocity_cmd : REAL := 0.011;   // Impreg Servo Operator Side Velocity Command
   p23_ao_servo_os_zero_offset : REAL := 0.036;   // Impreg Analog Outputs Drive Operator Side Servo Position Offset
   p23_ao_supply_selected_speed : REAL;   // Impreg Supply VFD Selected Speed
   p23_ave : CONTROL := (LEN := 9);   // Impreg Metering Roll VFD Avererage
   p23_cpr_gear_ratio : REAL := 91.4;
   p23_cpr_roll_diameter_ft : REAL := 0.833;
   p23_cpr_speed_to_vfd : SYS_SPEED_TO_VFD := (IN_gear_ratio := 91.4, IN_roll_diameter := 0.833);   // Impreg Outputs Speed to Impreg Pick Up Roll VFD
   p23_ctr_gear_ratio : REAL := 91.40625;
   p23_ctr_lfl_input_max : REAL := 30840.0;
   p23_ctr_lfl_input_min : REAL;
   p23_ctr_lfl_output_max : REAL := 100.0;
   p23_ctr_lfl_output_min : REAL;
   p23_ctr_roll_diameter_ft : REAL := 0.8333;
   p23_di_exhaust_speed_ok : BOOL;
   p23_di_filter_clean : BOOL := 1;
   p23_di_impreg_exhaust_running : BOOL;
   p23_di_impreg_tank_up : BOOL;   // Input Impreg Dip Tank Up
   p23_di_metering_bar_close : BOOL;   // Impreg Input SSS: Metering Bar Close
   p23_di_metering_bar_open : BOOL;   // Impreg Input SSS: Metering Bar Open
   p23_di_metering_roll : acs800_di_normal := (ready := 1, ctrl_from_net := 1, ref_from_net := 1, at_reference := 1);   // Impreg Digital Inputs Metering Roll VFD
   p23_di_servo_ds : servo_di := (mode_bit_1 := 1, homed := 1, stand_still := 1, drive_does_not_follow := 1, class_3_diagnostic := 1, operation_bit_15 := 1);   // Impreg Digital Inputs Servo Drive Side
   p23_di_servo_os : servo_di := (mode_bit_1 := 1, homed := 1, stand_still := 1, drive_does_not_follow := 1, class_3_diagnostic := 1, operation_bit_15 := 1);   // Impreg Digital Inputs Servo Operator Side
   p23_di_splice_jump : BOOL;   // Impreg Inputs PB: Splice Jump
   p23_di_spring : acs800_di_normal := (ready := 1, ctrl_from_net := 1, ref_from_net := 1, at_reference := 1);
   p23_di_srv_ds_ok : BOOL := 1;   // Impreg Inputs Metering Servo Drive Side Ok
   p23_di_srv_op_ok : BOOL := 1;   // Impreg Inputs Metering Servo Operator Side Ok
   p23_di_supply : acs800_di_normal := (ready := 1, ctrl_from_net := 1, ref_from_net := 1);   // Impreg Supply VFD VFD Inputs
   p23_di_supply_motor_therm : BOOL := 1;   // Impreg Inputs Supply Fan Motor Thermostat
   p23_di_supply_speed_ok : BOOL;
   p23_di_tank_level_high : BOOL;   // Impreg Input Dip Impreg Level High
   p23_di_tank_level_low : BOOL;   // Impreg Input Dip Impreg Level Low
   p23_di_therm : BOOL := 1;   // Impreg Inputs Metering Roll Motor Temperature Ok
   p23_di_though_level_low : BOOL;   // Impreg Input Dip Impreg Through Level Low
   p23_di_vfd_jog_fwd : BOOL;   // Impreg Input PB: VFD Jog FWD
   p23_di_vfd_jog_rev : BOOL;   // Impreg Input PB: VFD Jog REV
   p23_dint_to_hmi : DINT[17] := ([1] := 33845488, [3] := 207668736, [4] := 16, [5] := 2, [6] := 2, [7] := 3, [10] := -1, [11] := -1, [12] := -1, [13] := -1);   // Impreg Dint to HMI
        [0]   // Impreg Dint to HMI
        [0].0   // Impreg Dint to HMI Dip Tank Level Low
        [0].1   // Impreg Dint to HMI Through Level Low
        [0].2   // Impreg Dint to HMI Dip Tank Level High
        [0].3   // Imreg Dint to HMI PI: Exhaust Fan Running
        [0].16   // Impreg Dint to HMI PI: Exhaust & Supply Fan Started
        [0].18   // Impreg Dint to HMI PI: Dip Tank Up
        [1].0   // Impreg Dint to HMI Impreg Pickup Roll VFD Faulted
        [1].1   // Impreg Dint to HMI Impreg Pickup Roll VFD Warning
        [1].2   // Impreg Dint to HMI Impreg Pickup Roll VFD Running Forward
        [1].3   // Impreg Dint to HMI Impreg Pickup Roll VFD Running Reverse
        [1].4   // Impreg Dint to HMI Impreg Pickup Roll VFD Ready
        [1].5   // Impreg Dint to HMI Impreg Pickup Roll VFD Control from Net
        [1].6   // Impreg Dint to HMI Impreg Pickup Roll VFD Reference from Net
        [1].7   // Impreg Dint to HMI Impreg Pickup Roll VFD at Reference
        [1].8   // Impreg Dint to HMI Impreg Supply Fan VFD Faulted
        [1].9   // Impreg Dint to HMI Impreg Supply Fan VFD Warning
        [1].10   // Impreg Dint to HMI Impreg Supply Fan VFD Running Forward
        [1].11   // Impreg Dint to HMI Impreg Supply Fan VFD Running Reverse
        [1].12   // Impreg Dint to HMI Impreg Supply Fan VFD Ready
        [1].13   // Impreg Dint to HMI Impreg Supply Fan VFD Control from Net
        [1].14   // Impreg Dint to HMI Impreg Supply Fan VFD Reference from Net
        [1].15   // Impreg Dint to HMI Impreg Supply Fan VFD at Reference
        [1].16   // Impreg Dint to HMI PI: Servo Drive Side Not Ready
        [1].17   // Impreg Dint to HMI PI: Servo Drive Side BB Status
        [1].18   // Impreg Dint to HMI PI: Servo Drive Side AB Status
        [1].19   // Impreg Dint to HMI PI: Servo Drive Side AF Status
        [2]   // Impreg Dint to HMI
        [2].0   // Impreg Alarms A00: Supply VFD Faulted
        [2].1   // Impreg Alarms A01:
        [2].2   // Impreg Alarms A02: Supply VFD Drive Not Ready
        [2].3   // Impreg Alarms A03: Supply VFD Drive Not in Remote Mode
        [2].4   // Impreg Alarms A04: Supply VFD Motor Temperature
        [2].5   // Impreg Alarms A05:
        [2].6   // Impreg Alarms A06:
        [2].7   // Impreg Alarms A07:
        [2].8   // Impreg Alarms A08: Metering VFD Drive Fault
        [2].9   // Impreg Alarms A09:
        [2].10   // Impreg Alarms A10: Metering VFD Drive Not Ready
        [2].11   // Impreg Alarms A11: Metering VFD Drive Not in Remote Mode
        [2].12   // Impreg Alarms A12: Metering VFD Motor Temperature
        [2].13   // Impreg Alarms A13
        [2].14   // Impreg Alarms A14
        [2].15   // Impreg Alarms A15
        [2].16   // Impreg Alarms A16: Servo Drive Side Operation Mode Error
        [2].17   // Impreg Alarms A16: Servo Drive Side Faulted
        [2].20   // Impreg Alarms A20: Servo Operator Side Operation Mode Error
        [2].21   // Impreg Alarms A21: Servo Operator Side Faulted
        [2].22   // Impreg Alarms A22
        [2].23   // Impreg Alarms A23
        [2].24   // Impreg Alarms A24: LFL High High Alarm
        [2].25   // Impreg Alarms A25
        [2].26   // Impreg Alarms A26
        [2].27   // Impreg Alarms A27
        [2].28   // Impreg Alarms A28
        [2].29   // Impreg Alarms A29
        [2].30   // Impreg Alarms A30
        [2].31   // Impreg Alarms A31
        [3].8   // Impreg Dint to HMI Servo Drive Side Parameter Mode
        [3].9   // Impreg Dint to HMI Servo Drive Side Homed
        [3].10   // Impreg Dint to HMI Servo Drive Side Stand Still
        [3].11   // Impreg Dint to HMI Servo Drive Side At Target Position
        [3].12   // Impreg Dint to HMI Servo Drive Side Commmand Changed Bit
        [3].13   // Impreg Dint to HMI Servo Drive Side Operation Mode Error
        [3].14   // Impreg Dint to HMI Servo Drive Side Drive does not follow command value
        [3].15   // Impreg Dint to HMI Servo Drive Side Class 3 Diagnostic Message
        [3].16   // Impreg Dint to HMI Servo Drive Side Class 2 Diagnostic Message
        [3].17   // Impreg Dint to HMI Servo Drive Side Class 1 Diagnostic Message
        [3].20   // Impreg Dint to HMI Servo Operator Side Parameter Mode
        [3].21   // Impreg Dint to HMI Servo Operator Side Homed
        [3].22   // Impreg Dint to HMI Servo Operator Side Stand Still
        [3].23   // Impreg Dint to HMI Servo Operator Side At Target Position
        [3].24   // Impreg Dint to HMI Servo Operator Side Commmand Changed Bit
        [3].25   // Impreg Dint to HMI Servo Operator Side Operation Mode Error
        [3].26   // Impreg Dint to HMI Servo Operator Side Drive does not follow command value
        [3].27   // Impreg Dint to HMI Servo Operator Side Class 3 Diagnostic Message
        [3].28   // Impreg Dint to HMI Servo Operator Side Class 2 Diagnostic Message
        [3].29   // Impreg Dint to HMI Servo Operator Side Class 1 Diagnostic Message
        [4].0   // Impreg Warnings W00: Supply Fan VFD Drive Warning
        [4].1   // Impreg Warnings W01:
        [4].2   // Impreg Warnings W02:
        [4].3   // Impreg Warnings W03:
        [4].4   // Impreg Warnings W04: Metering VFD Drive Warning
        [4].5   // Impreg Warnings W05:
        [4].6   // Impreg Warnings W06:
        [4].7   // Impreg Warnings W07:
        [4].8   // Impreg Warnings W08: Servo Drive Side Warning
        [4].9   // Impreg Warnings W09:
        [4].10   // Impreg Warnings W10:
        [4].11   // Impreg Warnings W11:
        [4].12   // Impreg Warnings W12: Servo Operator Side Warning
        [4].13   // Impreg Warnings W13
        [4].14   // Impreg Warnings W14
        [4].15   // Impreg Warnings W15
        [4].16   // Impreg Warnings W16:
        [4].17   // Impreg Warnings W17
        [4].18   // Impreg Warnings W18
        [4].19   // Impreg Warnings W19
        [4].20   // Impreg Warnings W20
        [4].21   // Impreg Warnings W21
        [4].22   // Impreg Warnings W22
        [4].23   // Impreg Warnings W23
        [4].24   // Impreg Warnings W24: LFL High Warning
        [4].25   // Impreg Warnings W25
        [4].26   // Impreg Warnings W26
        [4].27   // Impreg Warnings W27
        [4].28   // Impreg Warnings W28
        [4].29   // Impreg Warnings W29
        [4].30   // Impreg Warnings W30
        [4].31   // Impreg Warnings W31
        [6]   // Imgreg Dint to HMI Servo Drive Side Status
   p23_do_enable_impreg_exhaust_fan : BOOL;   // Impreg Enclosure Digital Output Exhaust Fan Enable
   p23_do_enable_impreg_supply_fan : BOOL;   // Impreg Enclosure Digital Output Supply Fan Enable
   p23_do_impreg : acs800_do_normal;   // Impreg Digital Outputs VFD
   p23_do_impreg_nip_close : BOOL := 1;   // Impreg Digital Output Impreg Nip close
   p23_do_servo_ds : servo_do;   // Impreg Digital Outputs Drive Side Servo
   p23_do_servo_os : servo_do;   // Impreg Digital Outputs Operator Side Servo
   p23_do_Spring : acs800_do_normal;
   p23_do_supply : acs800_do_normal;   // Impreg Supply VFD] Outputs
   p23_mtr_acc_rate : REAL := 15.0;
   p23_mtr_decel_rate : REAL := 15.0;
   p23_param_lfl_hhl : REAL := 60.0;   // Impreg Parameter LFL High High Limit
   p23_param_lfl_hl : REAL := 10.0;   // Impreg Parameters LFL High Limit
   p23_param_min_start_tension : REAL := 20.0;
   p23_param_minus_adj_rate : REAL := -0.4;
   p23_param_mtr_jog_speed : REAL := 8.0;   // System Parameter Metering Roll Jog Speed
   p23_param_plus_adj_rate : REAL := 1.0;
   p23_param_servo_open_position : REAL := 0.011;
   p23_param_zone_pressure : REAL := -0.25;   // MOP HMI Iface Parameters Minimum Pressure
   p23_real_to_hmi : REAL[112] := ([0] := 0.018, [1] := 0.018, [2] := 0.005, [3] := 0.011, [8] := 3.8146973e-06, [11] := 60.0, [17] := 0.5, [22] := 0.0075000003, [23] := 65535.0, [27] := 1.6699092, [28] := -0.00967899, [55] := 10.0, [56] := 60.0, [58] := -0.25, [60] := 0.007, [61] := 0.007);   // Impreg Real to HMI
        [0]   // Impreg Real to HMI Servo Drive Side Offset
        [1]   // Impreg Real to HMI Servo Operator Side Offset
        [2]   // Impreg Real to HMI Servo Jog Velocity
        [3]   // Impreg Real to HMI Servo Positioning Velocity
        [6]   // Impreg Real to HMI Metering Roll VFD Speed
        [7]   // Impreg Real to HMI Metering Roll VFD Amps
        [8]   // Impreg Real to HMI Metering Roll VFD Hz
        [9]   // Impreg Real to HMI Supply Fan VFD RPM
        [10]   // Impreg Real to HMI Supply Fan VFD Amps
        [11]   // Impreg Real to HMI Supply Fan VFD Hz
        [60]   // Impreg Real to HMI Servo Drive Side Actual Position
        [61]   // Impreg Real to HMI Servo Operator Side Actual Position
   p23_servo_ds_error : SYS_ENC_WITH_ZERO_BIT := (OUT_Status := -1);   // Impreg Dint to HMI Servo Drive Side Error
   p23_servo_ds_warning : SYS_ENC_WITH_ZERO_BIT := (OUT_Status := -1);   // Impreg Dint to HMI Servo Drive Side Warning
   p23_servo_os_error : SYS_ENC_WITH_ZERO_BIT := (OUT_Status := -1);   // Impreg Dint to HMI Servo Operator Side Error
   p23_servo_os_warning : SYS_ENC_WITH_ZERO_BIT := (OUT_Status := -1);   // Impreg Dint to HMI Servo Operator Side Warning
   p23_spring_gear_ratio : REAL := 145.0;
   p23_spring_roll_diameter_ft : REAL := 0.5;
   p23_spring_speed_to_vfd : SYS_SPEED_TO_VFD := (IN_gear_ratio := 145.0, IN_roll_diameter := 0.5);
   p23r01 : routine := (comment := 7);   // Impreg Main
   p23r02 : routine := (comment := -1073741761, oneshot := 2);   // Impreg Misc Control
        .FAULT.0   // Impreg Misc Control Lower Flash Limit High High Limit Exceeded
        .WARNING.0   // Impreg Misc Control LFL Level Warning
        .UNACK_FAULT   // Impreg Misc Control Unacknoledged Faults Exist
        .UNACK_WARNING   // Impreg Misc Control Unacknowledged Warning Exists
   p23r02_fault_exists : BOOL;
   p23r02_open_pos_dint : DINT := 110;
   p23r02_open_pos_real : REAL := 0.011000001;
   p23r02_pb_start_exh : BOOL;
   p23r02_pb_stop_exh : BOOL;
   p23r02_request_nip_close : BOOL := 1;   // Impreg Misc Control Request Nip Close
   p23r02_timer_fault : TIMER[4] := ([0].PRE := 60, [1].PRE := 2000);   // Impreg Misc Control Timer Fault
   p23r02_timer_warning : TIMER[4] := ([1].PRE := 1000, [3].PRE := 5000);   // Impreg Misc Control Timer Warning
   p23r02_unack_fault : BOOL;   // Imperg Misc Control Unackn. Fault Exist
   p23r02_unack_warning : BOOL := 1;   // Impreg Misc Control Unackn. Warning Exist
   p23r02_warning_exists : BOOL := 1;
   p23r03 : routine := (comment := -1073741793);   // Impreg Inputs
        .WARNING.0   // Impreg Inputs Dip Tank Up and Oxidizer Not Ready
        .UNACK_FAULT   // Impreg Input Unacknoledged Faults Exist
        .UNACK_WARNING   // Impreg Input Unacknowledged Warning Exists
   p23r03_hz : SYS_SCP := (Input_Max := 1750.0, Output_Max := 60.0, Output := 3.8146973e-06);   // Impreg Roll Analog Inputs SCP Hz
   p23r03_impreg_lfl_monitor : SYS_SCP := (Input := 525.0, Input_Max := 30840.0, Output_Max := 100.0, Output := 1.7023346);   // Impreg Analog Inputs LFL Monitor Scaling
   p23r03_impreg_prs_input_max : REAL := 30840.0;
   p23r03_impreg_prs_input_min : REAL;
   p23r03_impreg_prs_output_max : REAL := 0.25;
   p23r03_impreg_prs_output_min : REAL := -0.25;
   p23r03_impreg_prs_scp : SYS_SCP := (Input := 14803.0, Input_Max := 30840.0, Output_Min := -0.25, Output_Max := 0.25, Output := -0.010003239);   // Impreg Analog Input Impreg Enclosure Pressure
   p23r03_metering_vfd_rpm_to_speed : SYS_RPM_TO_SPEED := (IN_gear_ratio := 91.40625, IN_roll_diameter := 0.8333);   // Impreg Metering Roll Input VFD AI
   p23r03_timer_fault : TIMER[4];   // Impreg Inputs Timer Fault
   p23r03_timer_warning : TIMER[4];   // Impreg Inputs Timer Warning
   p23r04 : routine := (comment := -1073741793);   // Impreg Outputs
        .UNACK_FAULT   // Impreg Output Unacknoledged Faults Exist
        .UNACK_WARNING   // Impreg Output Unacknowledged Warning Exists
   p23r04_timer_fault : TIMER[4];   // Impreg Outputs Fault Delay
   p23r04_timer_warning : TIMER[4];   // Impreg Outputs Warning Delay
   p23r05 : routine := (comment := -1073741761);   // Impreg Dint to HMI
        .UNACK_FAULT   // Impreg Dint to HMI Unacknoledged Faults Exist
        .UNACK_WARNING   // Impreg Dint to HMI Unacknowledged Warning Exists
   p23r05_supply_status : DINT := 3;
   p23r05_timer_fault : TIMER[4];   // Impreg Dint to HMI Timer Fault
   p23r05_timer_warning : TIMER[4];   // Impreg Dint to HMI Timer Warning
   p23r06 : routine := (comment := -1073741796);   // Impreg Real to HMI
        .UNACK_FAULT   // Impreg Real to HMI Unacknoledged Faults Exist
        .UNACK_WARNING   // Impreg Real to HMI Unacknowledged Warning Exists
   p23r06_timer_fault : TIMER[4];   // Impreg Real to HMI Fault Delay
   p23r06_timer_warning : TIMER[4];   // Impreg Real to HMI Warning Delay
   p23r07 : routine := (comment := -1073741761);   // Impreg Alarms
        .UNACK_FAULT   // Impreg Alarms Unacknoledged Faults Exist
        .UNACK_WARNING   // Impreg Alarms Unacknowledged Warning Exists
   p23r07_timer_fault : TIMER[4];   // Impreg Alarms Fault Delay
   p23r07_timer_warning : TIMER[4];   // Impreg Alarms Warning Delay
   p23r08 : routine := (comment := -1073741761);   // Impreg Warnings
        .UNACK_FAULT   // Impreg Warnings Unacknoledged Faults Exist
        .UNACK_WARNING   // Impreg Warnings Unacknowledged Warning Exists
   p23r08_timer_fault : TIMER[4];   // Impreg Warnings Fault Delay
   p23r08_timer_warning : TIMER[4];   // Impreg Warnings Warning Delay
   p23r09 : routine := (comment := -1073741761);   // Impreg Mode Selection
        .UNACK_FAULT   // Impreg Modes Unacknoledged Faults Exist
        .UNACK_WARNING   // Impreg Modes Unacknowledged Warning Exists
   p23r09_mode_run : BOOL := 1;   // Impreg Modes Pick Up Roll Run Mode
   p23r09_timer_fault : TIMER[4];   // Impreg Mode Selection Fault Delay
   p23r09_web_wet_ctrl_toggle : SYS_Toggle := (toggle_state := 1);   // Impreg Metering Roll VFD Web Wet Control
   p23r10 : routine := (comment := -1073741761);
   p23r10_timer_fault : TIMER[4];   // Impreg Parameters Fault Dwell Timer
   p23r10_timer_warning : TIMER[4];   // Impreg Parameters Warning Dwell Timer
   p23r11 : routine := (comment := -1073741570, state := 3);   // Impreg Servo Operator Side
        .FAULT.0   // Impreg Servo Opeator Side Operating Mode Error
        .FAULT.1   // Impreg Servo Operator Side Servo Fault
        .WARNING.0   // Impreg Servo Operator Side Servo Warning
